REGION Network 10: EM - UnHolding State Complete
   RUNG wire#powerrail
      Contact( "EM02".PackML_Sts.Alarm.sts_UnHolding_SC )
      wire#w1
      Contact( "EM02".PackML_Sts.CM01.sts_UnHolding_SC )
      wire#w2
      Contact( "EM02".PackML_Sts.CM02.sts_UnHolding_SC )
      wire#w3
      Contact( "EM02".PackML_Sts.CM03.sts_UnHolding_SC )
      wire#w4
      Contact( "EM02".PackML_Sts.CM04.sts_UnHolding_SC )
      wire#w5
      Contact( "EM02".PackML_Sts.CM05.sts_UnHolding_SC )
      wire#w6
      Contact( "EM02".PackML_Sts.CM06.sts_UnHolding_SC )
      wire#w7
      Contact( "EM02".PackML_Sts.CM07.sts_UnHolding_SC )
      wire#w8
      Contact( "EM02".PackML_Sts.CM08.sts_UnHolding_SC )
      wire#w9
      Contact( "EM02".PackML_Sts.CM09.sts_UnHolding_SC )
      wire#w10
      Contact( "EM02".PackML_Sts.CM10.sts_UnHolding_SC )
      wire#w11
      Coil( "EM02".PackML_Sts.Unit.sts_UnHolding_SC )
   END_RUNG
   RUNG wire#powerrail
      I_Contact( "EM02".PackML_Sts.Alarm.moduleActive )
   END_RUNG wire#w1
   RUNG wire#w1
      I_Contact( "EM02".PackML_Sts.CM01.moduleActive )
   END_RUNG wire#w2
   RUNG wire#w2
      I_Contact( "EM02".PackML_Sts.CM02.moduleActive )
   END_RUNG wire#w3
   RUNG wire#w3
      I_Contact( "EM02".PackML_Sts.CM03.moduleActive )
   END_RUNG wire#w4
   RUNG wire#w4
      I_Contact( "EM02".PackML_Sts.CM04.moduleActive )
   END_RUNG wire#w5
   RUNG wire#w5
      I_Contact( "EM02".PackML_Sts.CM05.moduleActive )
   END_RUNG wire#w6
   RUNG wire#w6
      I_Contact( "EM02".PackML_Sts.CM06.moduleActive )
   END_RUNG wire#w7
   RUNG wire#w7
      I_Contact( "EM02".PackML_Sts.CM07.moduleActive )
   END_RUNG wire#w8
   RUNG wire#w8
      I_Contact( "EM02".PackML_Sts.CM08.moduleActive )
   END_RUNG wire#w9
   RUNG wire#w9
      I_Contact( "EM02".PackML_Sts.CM09.moduleActive )
   END_RUNG wire#w10
   RUNG wire#w10
      I_Contact( "EM02".PackML_Sts.CM10.moduleActive )
   END_RUNG wire#w11
   // the same network as SCL:
   "EM02".PackML_Sts.Unit.sts_UnHolding_SC := ("EM02".PackML_Sts.Alarm.sts_UnHolding_SC OR NOT "EM02".PackML_Sts.Alarm.moduleActive) AND ("EM02".PackML_Sts.CM01.sts_UnHolding_SC OR NOT "EM02".PackML_Sts.CM01.moduleActive) AND ("EM02".PackML_Sts.CM02.sts_UnHolding_SC OR NOT "EM02".PackML_Sts.CM02.moduleActive) AND ("EM02".PackML_Sts.CM03.sts_UnHolding_SC OR NOT "EM02".PackML_Sts.CM03.moduleActive) AND ("EM02".PackML_Sts.CM04.sts_UnHolding_SC OR NOT "EM02".PackML_Sts.CM04.moduleActive) AND ("EM02".PackML_Sts.CM05.sts_UnHolding_SC OR NOT "EM02".PackML_Sts.CM05.moduleActive) AND ("EM02".PackML_Sts.CM06.sts_UnHolding_SC OR NOT "EM02".PackML_Sts.CM06.moduleActive) AND ("EM02".PackML_Sts.CM07.sts_UnHolding_SC OR NOT "EM02".PackML_Sts.CM07.moduleActive) AND ("EM02".PackML_Sts.CM08.sts_UnHolding_SC OR NOT "EM02".PackML_Sts.CM08.moduleActive) AND ("EM02".PackML_Sts.CM09.sts_UnHolding_SC OR NOT "EM02".PackML_Sts.CM09.moduleActive) AND ("EM02".PackML_Sts.CM10.sts_UnHolding_SC OR NOT "EM02".PackML_Sts.CM10.moduleActive);
END_REGION

REGION Network 11: EM - Suspend Command
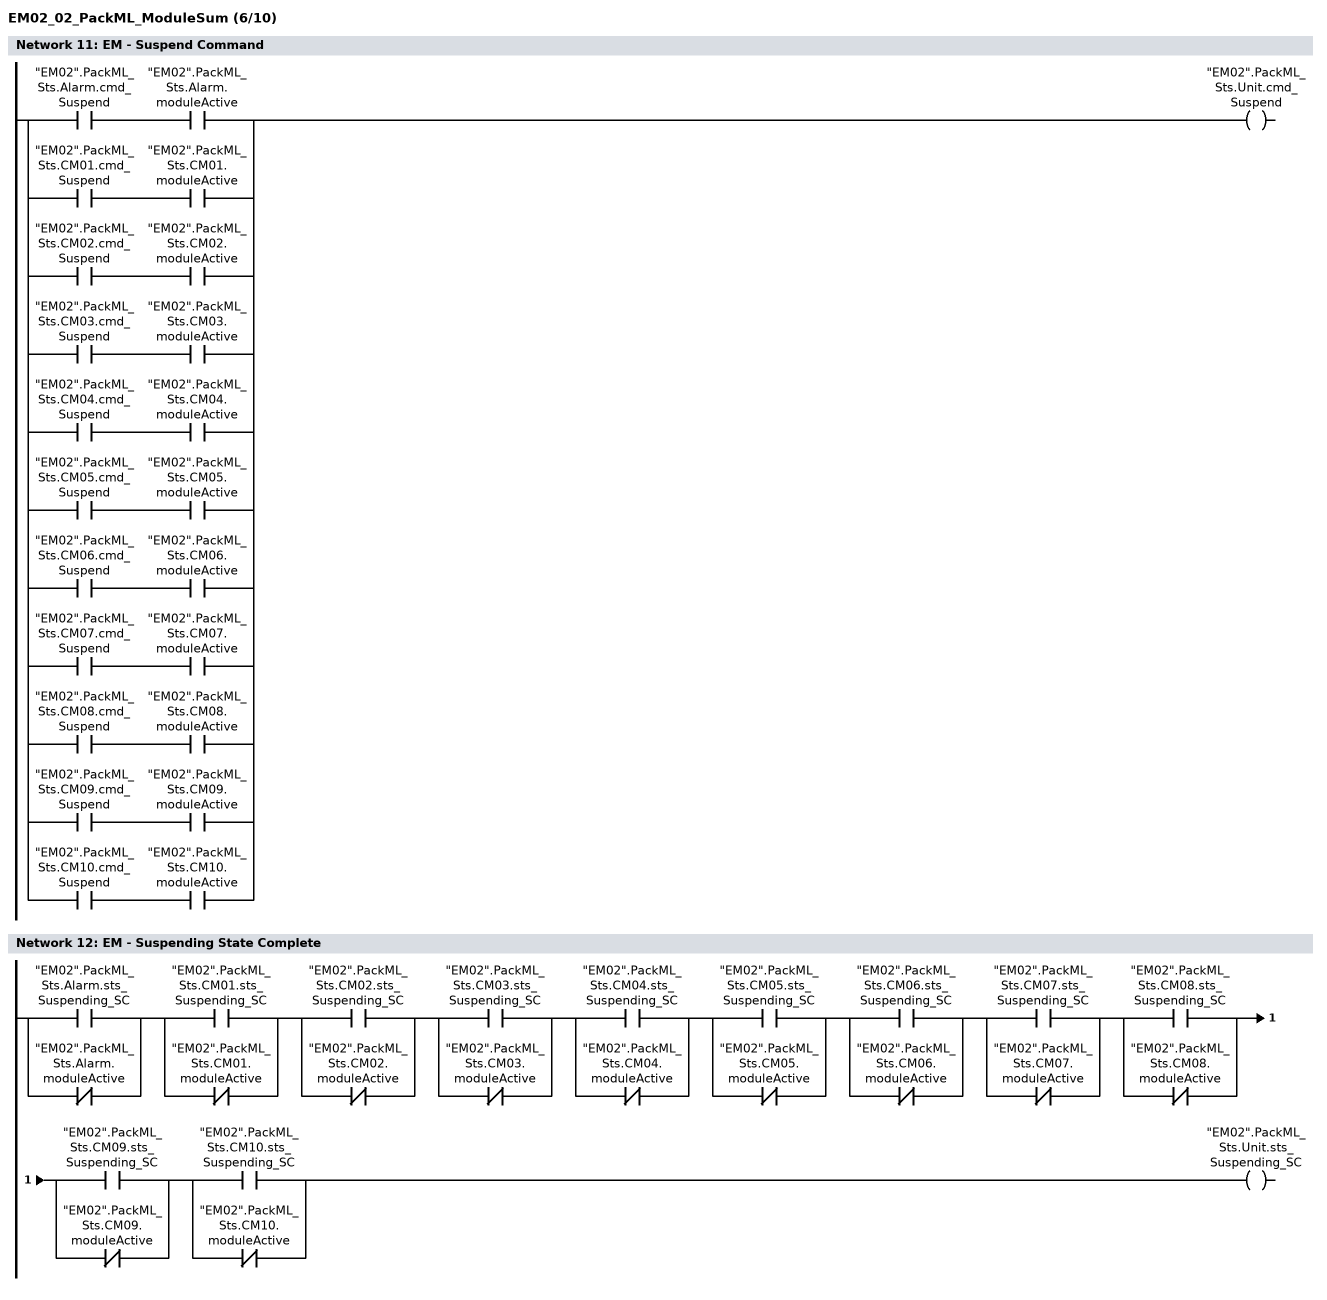
   RUNG wire#powerrail
      Contact( "EM02".PackML_Sts.Alarm.cmd_Suspend )
      Contact( "EM02".PackML_Sts.Alarm.moduleActive )
      wire#w1
      Coil( "EM02".PackML_Sts.Unit.cmd_Suspend )
   END_RUNG
   RUNG wire#powerrail
      Contact( "EM02".PackML_Sts.CM01.cmd_Suspend )
      Contact( "EM02".PackML_Sts.CM01.moduleActive )
   END_RUNG wire#w1
   RUNG wire#powerrail
      Contact( "EM02".PackML_Sts.CM02.cmd_Suspend )
      Contact( "EM02".PackML_Sts.CM02.moduleActive )
   END_RUNG wire#w1
   RUNG wire#powerrail
      Contact( "EM02".PackML_Sts.CM03.cmd_Suspend )
      Contact( "EM02".PackML_Sts.CM03.moduleActive )
   END_RUNG wire#w1
   RUNG wire#powerrail
      Contact( "EM02".PackML_Sts.CM04.cmd_Suspend )
      Contact( "EM02".PackML_Sts.CM04.moduleActive )
   END_RUNG wire#w1
   RUNG wire#powerrail
      Contact( "EM02".PackML_Sts.CM05.cmd_Suspend )
      Contact( "EM02".PackML_Sts.CM05.moduleActive )
   END_RUNG wire#w1
   RUNG wire#powerrail
      Contact( "EM02".PackML_Sts.CM06.cmd_Suspend )
      Contact( "EM02".PackML_Sts.CM06.moduleActive )
   END_RUNG wire#w1
   RUNG wire#powerrail
      Contact( "EM02".PackML_Sts.CM07.cmd_Suspend )
      Contact( "EM02".PackML_Sts.CM07.moduleActive )
   END_RUNG wire#w1
   RUNG wire#powerrail
      Contact( "EM02".PackML_Sts.CM08.cmd_Suspend )
      Contact( "EM02".PackML_Sts.CM08.moduleActive )
   END_RUNG wire#w1
   RUNG wire#powerrail
      Contact( "EM02".PackML_Sts.CM09.cmd_Suspend )
      Contact( "EM02".PackML_Sts.CM09.moduleActive )
   END_RUNG wire#w1
   RUNG wire#powerrail
      Contact( "EM02".PackML_Sts.CM10.cmd_Suspend )
      Contact( "EM02".PackML_Sts.CM10.moduleActive )
   END_RUNG wire#w1
   // the same network as SCL:
   "EM02".PackML_Sts.Unit.cmd_Suspend := ("EM02".PackML_Sts.Alarm.cmd_Suspend AND "EM02".PackML_Sts.Alarm.moduleActive) OR ("EM02".PackML_Sts.CM01.cmd_Suspend AND "EM02".PackML_Sts.CM01.moduleActive) OR ("EM02".PackML_Sts.CM02.cmd_Suspend AND "EM02".PackML_Sts.CM02.moduleActive) OR ("EM02".PackML_Sts.CM03.cmd_Suspend AND "EM02".PackML_Sts.CM03.moduleActive) OR ("EM02".PackML_Sts.CM04.cmd_Suspend AND "EM02".PackML_Sts.CM04.moduleActive) OR ("EM02".PackML_Sts.CM05.cmd_Suspend AND "EM02".PackML_Sts.CM05.moduleActive) OR ("EM02".PackML_Sts.CM06.cmd_Suspend AND "EM02".PackML_Sts.CM06.moduleActive) OR ("EM02".PackML_Sts.CM07.cmd_Suspend AND "EM02".PackML_Sts.CM07.moduleActive) OR ("EM02".PackML_Sts.CM08.cmd_Suspend AND "EM02".PackML_Sts.CM08.moduleActive) OR ("EM02".PackML_Sts.CM09.cmd_Suspend AND "EM02".PackML_Sts.CM09.moduleActive) OR ("EM02".PackML_Sts.CM10.cmd_Suspend AND "EM02".PackML_Sts.CM10.moduleActive);
END_REGION

REGION Network 12: EM - Suspending State Complete
   RUNG wire#powerrail
      Contact( "EM02".PackML_Sts.Alarm.sts_Suspending_SC )
      wire#w1
      Contact( "EM02".PackML_Sts.CM01.sts_Suspending_SC )
      wire#w2
      Contact( "EM02".PackML_Sts.CM02.sts_Suspending_SC )
      wire#w3
      Contact( "EM02".PackML_Sts.CM03.sts_Suspending_SC )
      wire#w4
      Contact( "EM02".PackML_Sts.CM04.sts_Suspending_SC )
      wire#w5
      Contact( "EM02".PackML_Sts.CM05.sts_Suspending_SC )
      wire#w6
      Contact( "EM02".PackML_Sts.CM06.sts_Suspending_SC )
      wire#w7
      Contact( "EM02".PackML_Sts.CM07.sts_Suspending_SC )
      wire#w8
      Contact( "EM02".PackML_Sts.CM08.sts_Suspending_SC )
      wire#w9
      Contact( "EM02".PackML_Sts.CM09.sts_Suspending_SC )
      wire#w10
      Contact( "EM02".PackML_Sts.CM10.sts_Suspending_SC )
      wire#w11
      Coil( "EM02".PackML_Sts.Unit.sts_Suspending_SC )
   END_RUNG
   RUNG wire#powerrail
      I_Contact( "EM02".PackML_Sts.Alarm.moduleActive )
   END_RUNG wire#w1
   RUNG wire#w1
      I_Contact( "EM02".PackML_Sts.CM01.moduleActive )
   END_RUNG wire#w2
   RUNG wire#w2
      I_Contact( "EM02".PackML_Sts.CM02.moduleActive )
   END_RUNG wire#w3
   RUNG wire#w3
      I_Contact( "EM02".PackML_Sts.CM03.moduleActive )
   END_RUNG wire#w4
   RUNG wire#w4
      I_Contact( "EM02".PackML_Sts.CM04.moduleActive )
   END_RUNG wire#w5
   RUNG wire#w5
      I_Contact( "EM02".PackML_Sts.CM05.moduleActive )
   END_RUNG wire#w6
   RUNG wire#w6
      I_Contact( "EM02".PackML_Sts.CM06.moduleActive )
   END_RUNG wire#w7
   RUNG wire#w7
      I_Contact( "EM02".PackML_Sts.CM07.moduleActive )
   END_RUNG wire#w8
   RUNG wire#w8
      I_Contact( "EM02".PackML_Sts.CM08.moduleActive )
   END_RUNG wire#w9
   RUNG wire#w9
      I_Contact( "EM02".PackML_Sts.CM09.moduleActive )
   END_RUNG wire#w10
   RUNG wire#w10
      I_Contact( "EM02".PackML_Sts.CM10.moduleActive )
   END_RUNG wire#w11
   // the same network as SCL:
   "EM02".PackML_Sts.Unit.sts_Suspending_SC := ("EM02".PackML_Sts.Alarm.sts_Suspending_SC OR NOT "EM02".PackML_Sts.Alarm.moduleActive) AND ("EM02".PackML_Sts.CM01.sts_Suspending_SC OR NOT "EM02".PackML_Sts.CM01.moduleActive) AND ("EM02".PackML_Sts.CM02.sts_Suspending_SC OR NOT "EM02".PackML_Sts.CM02.moduleActive) AND ("EM02".PackML_Sts.CM03.sts_Suspending_SC OR NOT "EM02".PackML_Sts.CM03.moduleActive) AND ("EM02".PackML_Sts.CM04.sts_Suspending_SC OR NOT "EM02".PackML_Sts.CM04.moduleActive) AND ("EM02".PackML_Sts.CM05.sts_Suspending_SC OR NOT "EM02".PackML_Sts.CM05.moduleActive) AND ("EM02".PackML_Sts.CM06.sts_Suspending_SC OR NOT "EM02".PackML_Sts.CM06.moduleActive) AND ("EM02".PackML_Sts.CM07.sts_Suspending_SC OR NOT "EM02".PackML_Sts.CM07.moduleActive) AND ("EM02".PackML_Sts.CM08.sts_Suspending_SC OR NOT "EM02".PackML_Sts.CM08.moduleActive) AND ("EM02".PackML_Sts.CM09.sts_Suspending_SC OR NOT "EM02".PackML_Sts.CM09.moduleActive) AND ("EM02".PackML_Sts.CM10.sts_Suspending_SC OR NOT "EM02".PackML_Sts.CM10.moduleActive);
END_REGION

REGION Network 13: EM - UnSuspend Command
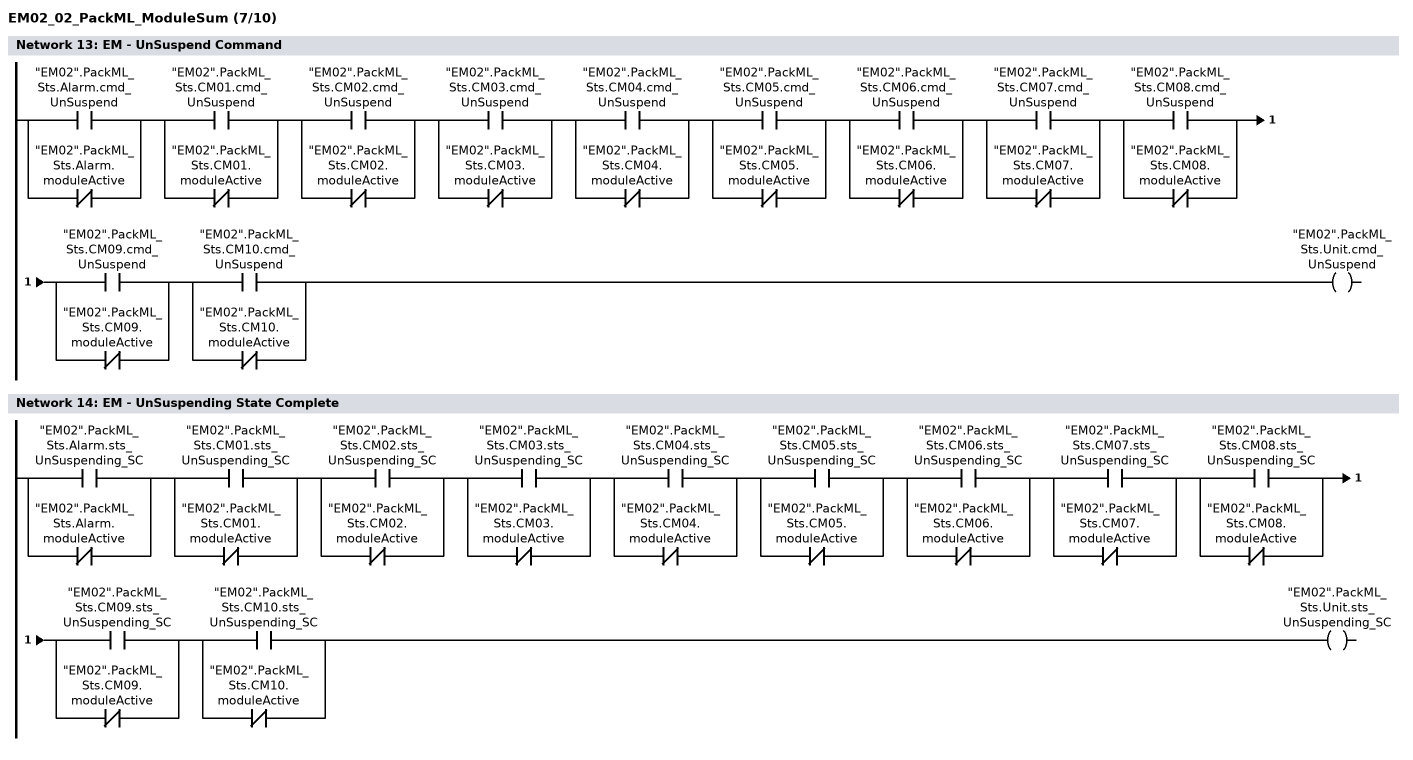
   RUNG wire#powerrail
      Contact( "EM02".PackML_Sts.Alarm.cmd_UnSuspend )
      wire#w1
      Contact( "EM02".PackML_Sts.CM01.cmd_UnSuspend )
      wire#w2
      Contact( "EM02".PackML_Sts.CM02.cmd_UnSuspend )
      wire#w3
      Contact( "EM02".PackML_Sts.CM03.cmd_UnSuspend )
      wire#w4
      Contact( "EM02".PackML_Sts.CM04.cmd_UnSuspend )
      wire#w5
      Contact( "EM02".PackML_Sts.CM05.cmd_UnSuspend )
      wire#w6
      Contact( "EM02".PackML_Sts.CM06.cmd_UnSuspend )
      wire#w7
      Contact( "EM02".PackML_Sts.CM07.cmd_UnSuspend )
      wire#w8
      Contact( "EM02".PackML_Sts.CM08.cmd_UnSuspend )
      wire#w9
      Contact( "EM02".PackML_Sts.CM09.cmd_UnSuspend )
      wire#w10
      Contact( "EM02".PackML_Sts.CM10.cmd_UnSuspend )
      wire#w11
      Coil( "EM02".PackML_Sts.Unit.cmd_UnSuspend )
   END_RUNG
   RUNG wire#powerrail
      I_Contact( "EM02".PackML_Sts.Alarm.moduleActive )
   END_RUNG wire#w1
   RUNG wire#w1
      I_Contact( "EM02".PackML_Sts.CM01.moduleActive )
   END_RUNG wire#w2
   RUNG wire#w2
      I_Contact( "EM02".PackML_Sts.CM02.moduleActive )
   END_RUNG wire#w3
   RUNG wire#w3
      I_Contact( "EM02".PackML_Sts.CM03.moduleActive )
   END_RUNG wire#w4
   RUNG wire#w4
      I_Contact( "EM02".PackML_Sts.CM04.moduleActive )
   END_RUNG wire#w5
   RUNG wire#w5
      I_Contact( "EM02".PackML_Sts.CM05.moduleActive )
   END_RUNG wire#w6
   RUNG wire#w6
      I_Contact( "EM02".PackML_Sts.CM06.moduleActive )
   END_RUNG wire#w7
   RUNG wire#w7
      I_Contact( "EM02".PackML_Sts.CM07.moduleActive )
   END_RUNG wire#w8
   RUNG wire#w8
      I_Contact( "EM02".PackML_Sts.CM08.moduleActive )
   END_RUNG wire#w9
   RUNG wire#w9
      I_Contact( "EM02".PackML_Sts.CM09.moduleActive )
   END_RUNG wire#w10
   RUNG wire#w10
      I_Contact( "EM02".PackML_Sts.CM10.moduleActive )
   END_RUNG wire#w11
   // the same network as SCL:
   "EM02".PackML_Sts.Unit.cmd_UnSuspend := ("EM02".PackML_Sts.Alarm.cmd_UnSuspend OR NOT "EM02".PackML_Sts.Alarm.moduleActive) AND ("EM02".PackML_Sts.CM01.cmd_UnSuspend OR NOT "EM02".PackML_Sts.CM01.moduleActive) AND ("EM02".PackML_Sts.CM02.cmd_UnSuspend OR NOT "EM02".PackML_Sts.CM02.moduleActive) AND ("EM02".PackML_Sts.CM03.cmd_UnSuspend OR NOT "EM02".PackML_Sts.CM03.moduleActive) AND ("EM02".PackML_Sts.CM04.cmd_UnSuspend OR NOT "EM02".PackML_Sts.CM04.moduleActive) AND ("EM02".PackML_Sts.CM05.cmd_UnSuspend OR NOT "EM02".PackML_Sts.CM05.moduleActive) AND ("EM02".PackML_Sts.CM06.cmd_UnSuspend OR NOT "EM02".PackML_Sts.CM06.moduleActive) AND ("EM02".PackML_Sts.CM07.cmd_UnSuspend OR NOT "EM02".PackML_Sts.CM07.moduleActive) AND ("EM02".PackML_Sts.CM08.cmd_UnSuspend OR NOT "EM02".PackML_Sts.CM08.moduleActive) AND ("EM02".PackML_Sts.CM09.cmd_UnSuspend OR NOT "EM02".PackML_Sts.CM09.moduleActive) AND ("EM02".PackML_Sts.CM10.cmd_UnSuspend OR NOT "EM02".PackML_Sts.CM10.moduleActive);
END_REGION

REGION Network 14: EM - UnSuspending State Complete
   RUNG wire#powerrail
      Contact( "EM02".PackML_Sts.Alarm.sts_UnSuspending_SC )
      wire#w1
      Contact( "EM02".PackML_Sts.CM01.sts_UnSuspending_SC )
      wire#w2
      Contact( "EM02".PackML_Sts.CM02.sts_UnSuspending_SC )
      wire#w3
      Contact( "EM02".PackML_Sts.CM03.sts_UnSuspending_SC )
      wire#w4
      Contact( "EM02".PackML_Sts.CM04.sts_UnSuspending_SC )
      wire#w5
      Contact( "EM02".PackML_Sts.CM05.sts_UnSuspending_SC )
      wire#w6
      Contact( "EM02".PackML_Sts.CM06.sts_UnSuspending_SC )
      wire#w7
      Contact( "EM02".PackML_Sts.CM07.sts_UnSuspending_SC )
      wire#w8
      Contact( "EM02".PackML_Sts.CM08.sts_UnSuspending_SC )
      wire#w9
      Contact( "EM02".PackML_Sts.CM09.sts_UnSuspending_SC )
      wire#w10
      Contact( "EM02".PackML_Sts.CM10.sts_UnSuspending_SC )
      wire#w11
      Coil( "EM02".PackML_Sts.Unit.sts_UnSuspending_SC )
   END_RUNG
   RUNG wire#powerrail
      I_Contact( "EM02".PackML_Sts.Alarm.moduleActive )
   END_RUNG wire#w1
   RUNG wire#w1
      I_Contact( "EM02".PackML_Sts.CM01.moduleActive )
   END_RUNG wire#w2
   RUNG wire#w2
      I_Contact( "EM02".PackML_Sts.CM02.moduleActive )
   END_RUNG wire#w3
   RUNG wire#w3
      I_Contact( "EM02".PackML_Sts.CM03.moduleActive )
   END_RUNG wire#w4
   RUNG wire#w4
      I_Contact( "EM02".PackML_Sts.CM04.moduleActive )
   END_RUNG wire#w5
   RUNG wire#w5
      I_Contact( "EM02".PackML_Sts.CM05.moduleActive )
   END_RUNG wire#w6
   RUNG wire#w6
      I_Contact( "EM02".PackML_Sts.CM06.moduleActive )
   END_RUNG wire#w7
   RUNG wire#w7
      I_Contact( "EM02".PackML_Sts.CM07.moduleActive )
   END_RUNG wire#w8
   RUNG wire#w8
      I_Contact( "EM02".PackML_Sts.CM08.moduleActive )
   END_RUNG wire#w9
   RUNG wire#w9
      I_Contact( "EM02".PackML_Sts.CM09.moduleActive )
   END_RUNG wire#w10
   RUNG wire#w10
      I_Contact( "EM02".PackML_Sts.CM10.moduleActive )
   END_RUNG wire#w11
   // the same network as SCL:
   "EM02".PackML_Sts.Unit.sts_UnSuspending_SC := ("EM02".PackML_Sts.Alarm.sts_UnSuspending_SC OR NOT "EM02".PackML_Sts.Alarm.moduleActive) AND ("EM02".PackML_Sts.CM01.sts_UnSuspending_SC OR NOT "EM02".PackML_Sts.CM01.moduleActive) AND ("EM02".PackML_Sts.CM02.sts_UnSuspending_SC OR NOT "EM02".PackML_Sts.CM02.moduleActive) AND ("EM02".PackML_Sts.CM03.sts_UnSuspending_SC OR NOT "EM02".PackML_Sts.CM03.moduleActive) AND ("EM02".PackML_Sts.CM04.sts_UnSuspending_SC OR NOT "EM02".PackML_Sts.CM04.moduleActive) AND ("EM02".PackML_Sts.CM05.sts_UnSuspending_SC OR NOT "EM02".PackML_Sts.CM05.moduleActive) AND ("EM02".PackML_Sts.CM06.sts_UnSuspending_SC OR NOT "EM02".PackML_Sts.CM06.moduleActive) AND ("EM02".PackML_Sts.CM07.sts_UnSuspending_SC OR NOT "EM02".PackML_Sts.CM07.moduleActive) AND ("EM02".PackML_Sts.CM08.sts_UnSuspending_SC OR NOT "EM02".PackML_Sts.CM08.moduleActive) AND ("EM02".PackML_Sts.CM09.sts_UnSuspending_SC OR NOT "EM02".PackML_Sts.CM09.moduleActive) AND ("EM02".PackML_Sts.CM10.sts_UnSuspending_SC OR NOT "EM02".PackML_Sts.CM10.moduleActive);
END_REGION

REGION Network 15: EM - Abort Command
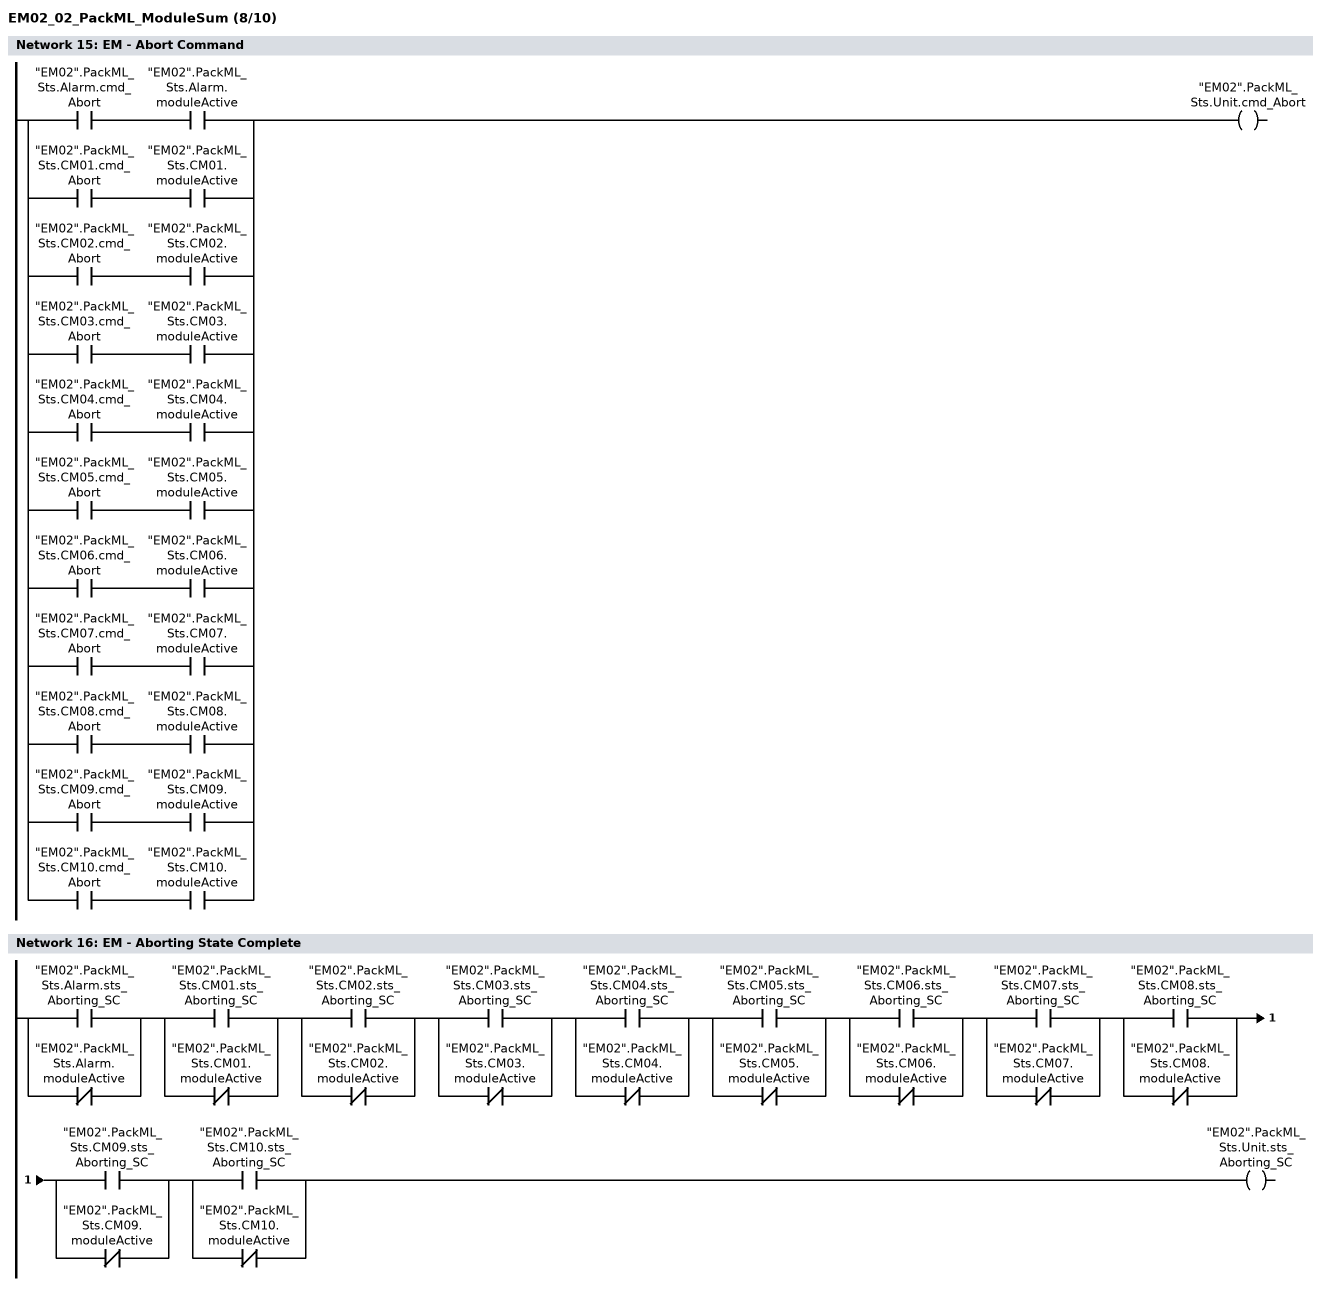
   RUNG wire#powerrail
      Contact( "EM02".PackML_Sts.Alarm.cmd_Abort )
      Contact( "EM02".PackML_Sts.Alarm.moduleActive )
      wire#w1
      Coil( "EM02".PackML_Sts.Unit.cmd_Abort )
   END_RUNG
   RUNG wire#powerrail
      Contact( "EM02".PackML_Sts.CM01.cmd_Abort )
      Contact( "EM02".PackML_Sts.CM01.moduleActive )
   END_RUNG wire#w1
   RUNG wire#powerrail
      Contact( "EM02".PackML_Sts.CM02.cmd_Abort )
      Contact( "EM02".PackML_Sts.CM02.moduleActive )
   END_RUNG wire#w1
   RUNG wire#powerrail
      Contact( "EM02".PackML_Sts.CM03.cmd_Abort )
      Contact( "EM02".PackML_Sts.CM03.moduleActive )
   END_RUNG wire#w1
   RUNG wire#powerrail
      Contact( "EM02".PackML_Sts.CM04.cmd_Abort )
      Contact( "EM02".PackML_Sts.CM04.moduleActive )
   END_RUNG wire#w1
   RUNG wire#powerrail
      Contact( "EM02".PackML_Sts.CM05.cmd_Abort )
      Contact( "EM02".PackML_Sts.CM05.moduleActive )
   END_RUNG wire#w1
   RUNG wire#powerrail
      Contact( "EM02".PackML_Sts.CM06.cmd_Abort )
      Contact( "EM02".PackML_Sts.CM06.moduleActive )
   END_RUNG wire#w1
   RUNG wire#powerrail
      Contact( "EM02".PackML_Sts.CM07.cmd_Abort )
      Contact( "EM02".PackML_Sts.CM07.moduleActive )
   END_RUNG wire#w1
   RUNG wire#powerrail
      Contact( "EM02".PackML_Sts.CM08.cmd_Abort )
      Contact( "EM02".PackML_Sts.CM08.moduleActive )
   END_RUNG wire#w1
   RUNG wire#powerrail
      Contact( "EM02".PackML_Sts.CM09.cmd_Abort )
      Contact( "EM02".PackML_Sts.CM09.moduleActive )
   END_RUNG wire#w1
   RUNG wire#powerrail
      Contact( "EM02".PackML_Sts.CM10.cmd_Abort )
      Contact( "EM02".PackML_Sts.CM10.moduleActive )
   END_RUNG wire#w1
   // the same network as SCL:
   "EM02".PackML_Sts.Unit.cmd_Abort := ("EM02".PackML_Sts.Alarm.cmd_Abort AND "EM02".PackML_Sts.Alarm.moduleActive) OR ("EM02".PackML_Sts.CM01.cmd_Abort AND "EM02".PackML_Sts.CM01.moduleActive) OR ("EM02".PackML_Sts.CM02.cmd_Abort AND "EM02".PackML_Sts.CM02.moduleActive) OR ("EM02".PackML_Sts.CM03.cmd_Abort AND "EM02".PackML_Sts.CM03.moduleActive) OR ("EM02".PackML_Sts.CM04.cmd_Abort AND "EM02".PackML_Sts.CM04.moduleActive) OR ("EM02".PackML_Sts.CM05.cmd_Abort AND "EM02".PackML_Sts.CM05.moduleActive) OR ("EM02".PackML_Sts.CM06.cmd_Abort AND "EM02".PackML_Sts.CM06.moduleActive) OR ("EM02".PackML_Sts.CM07.cmd_Abort AND "EM02".PackML_Sts.CM07.moduleActive) OR ("EM02".PackML_Sts.CM08.cmd_Abort AND "EM02".PackML_Sts.CM08.moduleActive) OR ("EM02".PackML_Sts.CM09.cmd_Abort AND "EM02".PackML_Sts.CM09.moduleActive) OR ("EM02".PackML_Sts.CM10.cmd_Abort AND "EM02".PackML_Sts.CM10.moduleActive);
END_REGION

REGION Network 16: EM - Aborting State Complete
   RUNG wire#powerrail
      Contact( "EM02".PackML_Sts.Alarm.sts_Aborting_SC )
      wire#w1
      Contact( "EM02".PackML_Sts.CM01.sts_Aborting_SC )
      wire#w2
      Contact( "EM02".PackML_Sts.CM02.sts_Aborting_SC )
      wire#w3
      Contact( "EM02".PackML_Sts.CM03.sts_Aborting_SC )
      wire#w4
      Contact( "EM02".PackML_Sts.CM04.sts_Aborting_SC )
      wire#w5
      Contact( "EM02".PackML_Sts.CM05.sts_Aborting_SC )
      wire#w6
      Contact( "EM02".PackML_Sts.CM06.sts_Aborting_SC )
      wire#w7
      Contact( "EM02".PackML_Sts.CM07.sts_Aborting_SC )
      wire#w8
      Contact( "EM02".PackML_Sts.CM08.sts_Aborting_SC )
      wire#w9
      Contact( "EM02".PackML_Sts.CM09.sts_Aborting_SC )
      wire#w10
      Contact( "EM02".PackML_Sts.CM10.sts_Aborting_SC )
      wire#w11
      Coil( "EM02".PackML_Sts.Unit.sts_Aborting_SC )
   END_RUNG
   RUNG wire#powerrail
      I_Contact( "EM02".PackML_Sts.Alarm.moduleActive )
   END_RUNG wire#w1
   RUNG wire#w1
      I_Contact( "EM02".PackML_Sts.CM01.moduleActive )
   END_RUNG wire#w2
   RUNG wire#w2
      I_Contact( "EM02".PackML_Sts.CM02.moduleActive )
   END_RUNG wire#w3
   RUNG wire#w3
      I_Contact( "EM02".PackML_Sts.CM03.moduleActive )
   END_RUNG wire#w4
   RUNG wire#w4
      I_Contact( "EM02".PackML_Sts.CM04.moduleActive )
   END_RUNG wire#w5
   RUNG wire#w5
      I_Contact( "EM02".PackML_Sts.CM05.moduleActive )
   END_RUNG wire#w6
   RUNG wire#w6
      I_Contact( "EM02".PackML_Sts.CM06.moduleActive )
   END_RUNG wire#w7
   RUNG wire#w7
      I_Contact( "EM02".PackML_Sts.CM07.moduleActive )
   END_RUNG wire#w8
   RUNG wire#w8
      I_Contact( "EM02".PackML_Sts.CM08.moduleActive )
   END_RUNG wire#w9
   RUNG wire#w9
      I_Contact( "EM02".PackML_Sts.CM09.moduleActive )
   END_RUNG wire#w10
   RUNG wire#w10
      I_Contact( "EM02".PackML_Sts.CM10.moduleActive )
   END_RUNG wire#w11
   // the same network as SCL:
   "EM02".PackML_Sts.Unit.sts_Aborting_SC := ("EM02".PackML_Sts.Alarm.sts_Aborting_SC OR NOT "EM02".PackML_Sts.Alarm.moduleActive) AND ("EM02".PackML_Sts.CM01.sts_Aborting_SC OR NOT "EM02".PackML_Sts.CM01.moduleActive) AND ("EM02".PackML_Sts.CM02.sts_Aborting_SC OR NOT "EM02".PackML_Sts.CM02.moduleActive) AND ("EM02".PackML_Sts.CM03.sts_Aborting_SC OR NOT "EM02".PackML_Sts.CM03.moduleActive) AND ("EM02".PackML_Sts.CM04.sts_Aborting_SC OR NOT "EM02".PackML_Sts.CM04.moduleActive) AND ("EM02".PackML_Sts.CM05.sts_Aborting_SC OR NOT "EM02".PackML_Sts.CM05.moduleActive) AND ("EM02".PackML_Sts.CM06.sts_Aborting_SC OR NOT "EM02".PackML_Sts.CM06.moduleActive) AND ("EM02".PackML_Sts.CM07.sts_Aborting_SC OR NOT "EM02".PackML_Sts.CM07.moduleActive) AND ("EM02".PackML_Sts.CM08.sts_Aborting_SC OR NOT "EM02".PackML_Sts.CM08.moduleActive) AND ("EM02".PackML_Sts.CM09.sts_Aborting_SC OR NOT "EM02".PackML_Sts.CM09.moduleActive) AND ("EM02".PackML_Sts.CM10.sts_Aborting_SC OR NOT "EM02".PackML_Sts.CM10.moduleActive);
END_REGION

REGION Network 17: EM - Clear Command
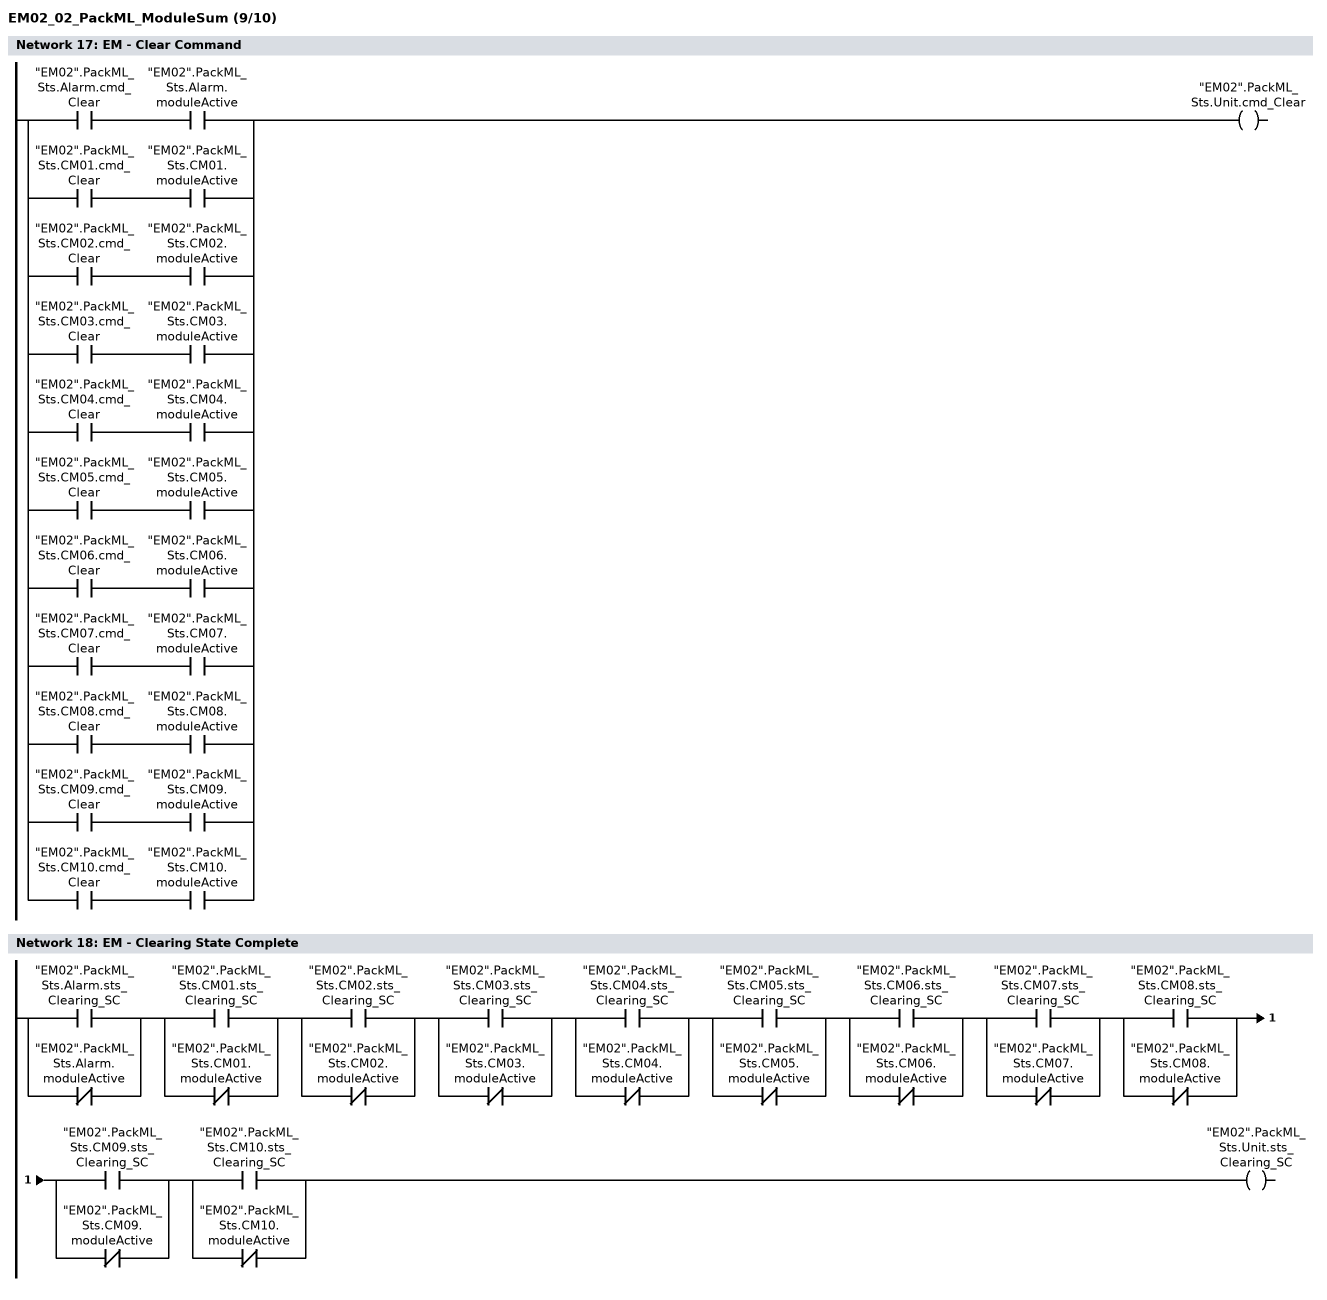
   RUNG wire#powerrail
      Contact( "EM02".PackML_Sts.Alarm.cmd_Clear )
      Contact( "EM02".PackML_Sts.Alarm.moduleActive )
      wire#w1
      Coil( "EM02".PackML_Sts.Unit.cmd_Clear )
   END_RUNG
   RUNG wire#powerrail
      Contact( "EM02".PackML_Sts.CM01.cmd_Clear )
      Contact( "EM02".PackML_Sts.CM01.moduleActive )
   END_RUNG wire#w1
   RUNG wire#powerrail
      Contact( "EM02".PackML_Sts.CM02.cmd_Clear )
      Contact( "EM02".PackML_Sts.CM02.moduleActive )
   END_RUNG wire#w1
   RUNG wire#powerrail
      Contact( "EM02".PackML_Sts.CM03.cmd_Clear )
      Contact( "EM02".PackML_Sts.CM03.moduleActive )
   END_RUNG wire#w1
   RUNG wire#powerrail
      Contact( "EM02".PackML_Sts.CM04.cmd_Clear )
      Contact( "EM02".PackML_Sts.CM04.moduleActive )
   END_RUNG wire#w1
   RUNG wire#powerrail
      Contact( "EM02".PackML_Sts.CM05.cmd_Clear )
      Contact( "EM02".PackML_Sts.CM05.moduleActive )
   END_RUNG wire#w1
   RUNG wire#powerrail
      Contact( "EM02".PackML_Sts.CM06.cmd_Clear )
      Contact( "EM02".PackML_Sts.CM06.moduleActive )
   END_RUNG wire#w1
   RUNG wire#powerrail
      Contact( "EM02".PackML_Sts.CM07.cmd_Clear )
      Contact( "EM02".PackML_Sts.CM07.moduleActive )
   END_RUNG wire#w1
   RUNG wire#powerrail
      Contact( "EM02".PackML_Sts.CM08.cmd_Clear )
      Contact( "EM02".PackML_Sts.CM08.moduleActive )
   END_RUNG wire#w1
   RUNG wire#powerrail
      Contact( "EM02".PackML_Sts.CM09.cmd_Clear )
      Contact( "EM02".PackML_Sts.CM09.moduleActive )
   END_RUNG wire#w1
   RUNG wire#powerrail
      Contact( "EM02".PackML_Sts.CM10.cmd_Clear )
      Contact( "EM02".PackML_Sts.CM10.moduleActive )
   END_RUNG wire#w1
   // the same network as SCL:
   "EM02".PackML_Sts.Unit.cmd_Clear := ("EM02".PackML_Sts.Alarm.cmd_Clear AND "EM02".PackML_Sts.Alarm.moduleActive) OR ("EM02".PackML_Sts.CM01.cmd_Clear AND "EM02".PackML_Sts.CM01.moduleActive) OR ("EM02".PackML_Sts.CM02.cmd_Clear AND "EM02".PackML_Sts.CM02.moduleActive) OR ("EM02".PackML_Sts.CM03.cmd_Clear AND "EM02".PackML_Sts.CM03.moduleActive) OR ("EM02".PackML_Sts.CM04.cmd_Clear AND "EM02".PackML_Sts.CM04.moduleActive) OR ("EM02".PackML_Sts.CM05.cmd_Clear AND "EM02".PackML_Sts.CM05.moduleActive) OR ("EM02".PackML_Sts.CM06.cmd_Clear AND "EM02".PackML_Sts.CM06.moduleActive) OR ("EM02".PackML_Sts.CM07.cmd_Clear AND "EM02".PackML_Sts.CM07.moduleActive) OR ("EM02".PackML_Sts.CM08.cmd_Clear AND "EM02".PackML_Sts.CM08.moduleActive) OR ("EM02".PackML_Sts.CM09.cmd_Clear AND "EM02".PackML_Sts.CM09.moduleActive) OR ("EM02".PackML_Sts.CM10.cmd_Clear AND "EM02".PackML_Sts.CM10.moduleActive);
END_REGION

REGION Network 18: EM - Clearing State Complete
   RUNG wire#powerrail
      Contact( "EM02".PackML_Sts.Alarm.sts_Clearing_SC )
      wire#w1
      Contact( "EM02".PackML_Sts.CM01.sts_Clearing_SC )
      wire#w2
      Contact( "EM02".PackML_Sts.CM02.sts_Clearing_SC )
      wire#w3
      Contact( "EM02".PackML_Sts.CM03.sts_Clearing_SC )
      wire#w4
      Contact( "EM02".PackML_Sts.CM04.sts_Clearing_SC )
      wire#w5
      Contact( "EM02".PackML_Sts.CM05.sts_Clearing_SC )
      wire#w6
      Contact( "EM02".PackML_Sts.CM06.sts_Clearing_SC )
      wire#w7
      Contact( "EM02".PackML_Sts.CM07.sts_Clearing_SC )
      wire#w8
      Contact( "EM02".PackML_Sts.CM08.sts_Clearing_SC )
      wire#w9
      Contact( "EM02".PackML_Sts.CM09.sts_Clearing_SC )
      wire#w10
      Contact( "EM02".PackML_Sts.CM10.sts_Clearing_SC )
      wire#w11
      Coil( "EM02".PackML_Sts.Unit.sts_Clearing_SC )
   END_RUNG
   RUNG wire#powerrail
      I_Contact( "EM02".PackML_Sts.Alarm.moduleActive )
   END_RUNG wire#w1
   RUNG wire#w1
      I_Contact( "EM02".PackML_Sts.CM01.moduleActive )
   END_RUNG wire#w2
   RUNG wire#w2
      I_Contact( "EM02".PackML_Sts.CM02.moduleActive )
   END_RUNG wire#w3
   RUNG wire#w3
      I_Contact( "EM02".PackML_Sts.CM03.moduleActive )
   END_RUNG wire#w4
   RUNG wire#w4
      I_Contact( "EM02".PackML_Sts.CM04.moduleActive )
   END_RUNG wire#w5
   RUNG wire#w5
      I_Contact( "EM02".PackML_Sts.CM05.moduleActive )
   END_RUNG wire#w6
   RUNG wire#w6
      I_Contact( "EM02".PackML_Sts.CM06.moduleActive )
   END_RUNG wire#w7
   RUNG wire#w7
      I_Contact( "EM02".PackML_Sts.CM07.moduleActive )
   END_RUNG wire#w8
   RUNG wire#w8
      I_Contact( "EM02".PackML_Sts.CM08.moduleActive )
   END_RUNG wire#w9
   RUNG wire#w9
      I_Contact( "EM02".PackML_Sts.CM09.moduleActive )
   END_RUNG wire#w10
   RUNG wire#w10
      I_Contact( "EM02".PackML_Sts.CM10.moduleActive )
   END_RUNG wire#w11
   // the same network as SCL:
   "EM02".PackML_Sts.Unit.sts_Clearing_SC := ("EM02".PackML_Sts.Alarm.sts_Clearing_SC OR NOT "EM02".PackML_Sts.Alarm.moduleActive) AND ("EM02".PackML_Sts.CM01.sts_Clearing_SC OR NOT "EM02".PackML_Sts.CM01.moduleActive) AND ("EM02".PackML_Sts.CM02.sts_Clearing_SC OR NOT "EM02".PackML_Sts.CM02.moduleActive) AND ("EM02".PackML_Sts.CM03.sts_Clearing_SC OR NOT "EM02".PackML_Sts.CM03.moduleActive) AND ("EM02".PackML_Sts.CM04.sts_Clearing_SC OR NOT "EM02".PackML_Sts.CM04.moduleActive) AND ("EM02".PackML_Sts.CM05.sts_Clearing_SC OR NOT "EM02".PackML_Sts.CM05.moduleActive) AND ("EM02".PackML_Sts.CM06.sts_Clearing_SC OR NOT "EM02".PackML_Sts.CM06.moduleActive) AND ("EM02".PackML_Sts.CM07.sts_Clearing_SC OR NOT "EM02".PackML_Sts.CM07.moduleActive) AND ("EM02".PackML_Sts.CM08.sts_Clearing_SC OR NOT "EM02".PackML_Sts.CM08.moduleActive) AND ("EM02".PackML_Sts.CM09.sts_Clearing_SC OR NOT "EM02".PackML_Sts.CM09.moduleActive) AND ("EM02".PackML_Sts.CM10.sts_Clearing_SC OR NOT "EM02".PackML_Sts.CM10.moduleActive);
END_REGION

REGION Network 19: EM - Execute State Complete
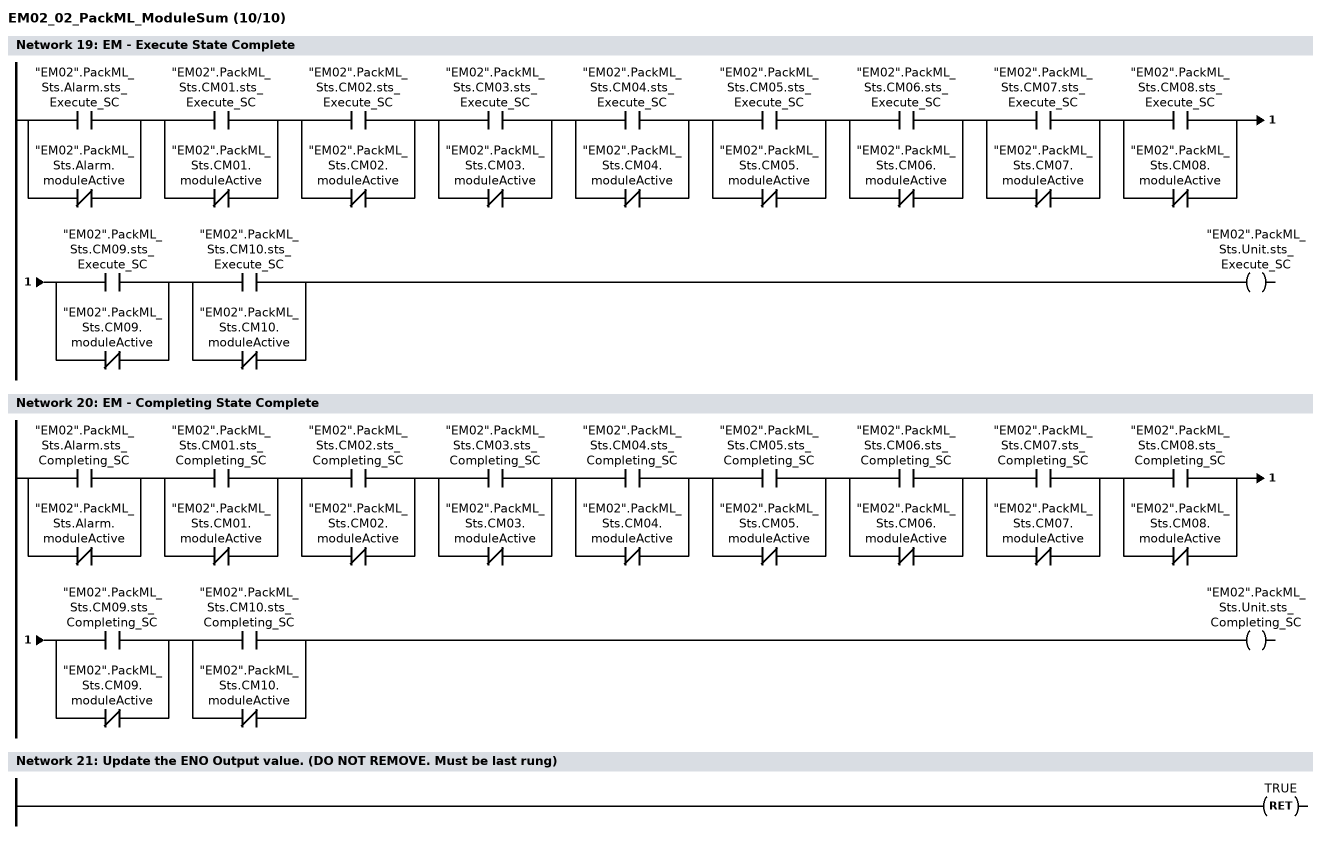
   RUNG wire#powerrail
      Contact( "EM02".PackML_Sts.Alarm.sts_Execute_SC )
      wire#w1
      Contact( "EM02".PackML_Sts.CM01.sts_Execute_SC )
      wire#w2
      Contact( "EM02".PackML_Sts.CM02.sts_Execute_SC )
      wire#w3
      Contact( "EM02".PackML_Sts.CM03.sts_Execute_SC )
      wire#w4
      Contact( "EM02".PackML_Sts.CM04.sts_Execute_SC )
      wire#w5
      Contact( "EM02".PackML_Sts.CM05.sts_Execute_SC )
      wire#w6
      Contact( "EM02".PackML_Sts.CM06.sts_Execute_SC )
      wire#w7
      Contact( "EM02".PackML_Sts.CM07.sts_Execute_SC )
      wire#w8
      Contact( "EM02".PackML_Sts.CM08.sts_Execute_SC )
      wire#w9
      Contact( "EM02".PackML_Sts.CM09.sts_Execute_SC )
      wire#w10
      Contact( "EM02".PackML_Sts.CM10.sts_Execute_SC )
      wire#w11
      Coil( "EM02".PackML_Sts.Unit.sts_Execute_SC )
   END_RUNG
   RUNG wire#powerrail
      I_Contact( "EM02".PackML_Sts.Alarm.moduleActive )
   END_RUNG wire#w1
   RUNG wire#w1
      I_Contact( "EM02".PackML_Sts.CM01.moduleActive )
   END_RUNG wire#w2
   RUNG wire#w2
      I_Contact( "EM02".PackML_Sts.CM02.moduleActive )
   END_RUNG wire#w3
   RUNG wire#w3
      I_Contact( "EM02".PackML_Sts.CM03.moduleActive )
   END_RUNG wire#w4
   RUNG wire#w4
      I_Contact( "EM02".PackML_Sts.CM04.moduleActive )
   END_RUNG wire#w5
   RUNG wire#w5
      I_Contact( "EM02".PackML_Sts.CM05.moduleActive )
   END_RUNG wire#w6
   RUNG wire#w6
      I_Contact( "EM02".PackML_Sts.CM06.moduleActive )
   END_RUNG wire#w7
   RUNG wire#w7
      I_Contact( "EM02".PackML_Sts.CM07.moduleActive )
   END_RUNG wire#w8
   RUNG wire#w8
      I_Contact( "EM02".PackML_Sts.CM08.moduleActive )
   END_RUNG wire#w9
   RUNG wire#w9
      I_Contact( "EM02".PackML_Sts.CM09.moduleActive )
   END_RUNG wire#w10
   RUNG wire#w10
      I_Contact( "EM02".PackML_Sts.CM10.moduleActive )
   END_RUNG wire#w11
   // the same network as SCL:
   "EM02".PackML_Sts.Unit.sts_Execute_SC := ("EM02".PackML_Sts.Alarm.sts_Execute_SC OR NOT "EM02".PackML_Sts.Alarm.moduleActive) AND ("EM02".PackML_Sts.CM01.sts_Execute_SC OR NOT "EM02".PackML_Sts.CM01.moduleActive) AND ("EM02".PackML_Sts.CM02.sts_Execute_SC OR NOT "EM02".PackML_Sts.CM02.moduleActive) AND ("EM02".PackML_Sts.CM03.sts_Execute_SC OR NOT "EM02".PackML_Sts.CM03.moduleActive) AND ("EM02".PackML_Sts.CM04.sts_Execute_SC OR NOT "EM02".PackML_Sts.CM04.moduleActive) AND ("EM02".PackML_Sts.CM05.sts_Execute_SC OR NOT "EM02".PackML_Sts.CM05.moduleActive) AND ("EM02".PackML_Sts.CM06.sts_Execute_SC OR NOT "EM02".PackML_Sts.CM06.moduleActive) AND ("EM02".PackML_Sts.CM07.sts_Execute_SC OR NOT "EM02".PackML_Sts.CM07.moduleActive) AND ("EM02".PackML_Sts.CM08.sts_Execute_SC OR NOT "EM02".PackML_Sts.CM08.moduleActive) AND ("EM02".PackML_Sts.CM09.sts_Execute_SC OR NOT "EM02".PackML_Sts.CM09.moduleActive) AND ("EM02".PackML_Sts.CM10.sts_Execute_SC OR NOT "EM02".PackML_Sts.CM10.moduleActive);
END_REGION

REGION Network 20: EM - Completing State Complete
   RUNG wire#powerrail
      Contact( "EM02".PackML_Sts.Alarm.sts_Completing_SC )
      wire#w1
      Contact( "EM02".PackML_Sts.CM01.sts_Completing_SC )
      wire#w2
      Contact( "EM02".PackML_Sts.CM02.sts_Completing_SC )
      wire#w3
      Contact( "EM02".PackML_Sts.CM03.sts_Completing_SC )
      wire#w4
      Contact( "EM02".PackML_Sts.CM04.sts_Completing_SC )
      wire#w5
      Contact( "EM02".PackML_Sts.CM05.sts_Completing_SC )
      wire#w6
      Contact( "EM02".PackML_Sts.CM06.sts_Completing_SC )
      wire#w7
      Contact( "EM02".PackML_Sts.CM07.sts_Completing_SC )
      wire#w8
      Contact( "EM02".PackML_Sts.CM08.sts_Completing_SC )
      wire#w9
      Contact( "EM02".PackML_Sts.CM09.sts_Completing_SC )
      wire#w10
      Contact( "EM02".PackML_Sts.CM10.sts_Completing_SC )
      wire#w11
      Coil( "EM02".PackML_Sts.Unit.sts_Completing_SC )
   END_RUNG
   RUNG wire#powerrail
      I_Contact( "EM02".PackML_Sts.Alarm.moduleActive )
   END_RUNG wire#w1
   RUNG wire#w1
      I_Contact( "EM02".PackML_Sts.CM01.moduleActive )
   END_RUNG wire#w2
   RUNG wire#w2
      I_Contact( "EM02".PackML_Sts.CM02.moduleActive )
   END_RUNG wire#w3
   RUNG wire#w3
      I_Contact( "EM02".PackML_Sts.CM03.moduleActive )
   END_RUNG wire#w4
   RUNG wire#w4
      I_Contact( "EM02".PackML_Sts.CM04.moduleActive )
   END_RUNG wire#w5
   RUNG wire#w5
      I_Contact( "EM02".PackML_Sts.CM05.moduleActive )
   END_RUNG wire#w6
   RUNG wire#w6
      I_Contact( "EM02".PackML_Sts.CM06.moduleActive )
   END_RUNG wire#w7
   RUNG wire#w7
      I_Contact( "EM02".PackML_Sts.CM07.moduleActive )
   END_RUNG wire#w8
   RUNG wire#w8
      I_Contact( "EM02".PackML_Sts.CM08.moduleActive )
   END_RUNG wire#w9
   RUNG wire#w9
      I_Contact( "EM02".PackML_Sts.CM09.moduleActive )
   END_RUNG wire#w10
   RUNG wire#w10
      I_Contact( "EM02".PackML_Sts.CM10.moduleActive )
   END_RUNG wire#w11
   // the same network as SCL:
   "EM02".PackML_Sts.Unit.sts_Completing_SC := ("EM02".PackML_Sts.Alarm.sts_Completing_SC OR NOT "EM02".PackML_Sts.Alarm.moduleActive) AND ("EM02".PackML_Sts.CM01.sts_Completing_SC OR NOT "EM02".PackML_Sts.CM01.moduleActive) AND ("EM02".PackML_Sts.CM02.sts_Completing_SC OR NOT "EM02".PackML_Sts.CM02.moduleActive) AND ("EM02".PackML_Sts.CM03.sts_Completing_SC OR NOT "EM02".PackML_Sts.CM03.moduleActive) AND ("EM02".PackML_Sts.CM04.sts_Completing_SC OR NOT "EM02".PackML_Sts.CM04.moduleActive) AND ("EM02".PackML_Sts.CM05.sts_Completing_SC OR NOT "EM02".PackML_Sts.CM05.moduleActive) AND ("EM02".PackML_Sts.CM06.sts_Completing_SC OR NOT "EM02".PackML_Sts.CM06.moduleActive) AND ("EM02".PackML_Sts.CM07.sts_Completing_SC OR NOT "EM02".PackML_Sts.CM07.moduleActive) AND ("EM02".PackML_Sts.CM08.sts_Completing_SC OR NOT "EM02".PackML_Sts.CM08.moduleActive) AND ("EM02".PackML_Sts.CM09.sts_Completing_SC OR NOT "EM02".PackML_Sts.CM09.moduleActive) AND ("EM02".PackML_Sts.CM10.sts_Completing_SC OR NOT "EM02".PackML_Sts.CM10.moduleActive);
END_REGION

REGION Network 21: Update the ENO Output value. (DO NOT REMOVE. Must be last rung)
   RUNG wire#powerrail
      ReturnCoil( TRUE )
   END_RUNG
   // the same network as SCL:
   ENO := TRUE;
   RETURN;
END_REGION
END_FUNCTION_BLOCK

ORGANIZATION_BLOCK "COMPLETE RESTART"   // OB100, LAD, Startup
TITLE = "Complete Restart"
{ S7_Optimized_Access := 'TRUE' }
VERSION : 0.1
// stored: AutoNumber true, IsIECCheckEnabled false, SetENOAutomatically false
   VAR_INPUT
      LostRetentive : Bool;   // True if retentive data are lost
      LostRTC : Bool;   // True if date and time are lost
   END_VAR
BEGIN
END_ORGANIZATION_BLOCK

ORGANIZATION_BLOCK "CYC_INT5"   // OB35, LAD, CyclicInterrupt
TITLE = "Cyclic Interrupt"
{ S7_Optimized_Access := 'TRUE' }
VERSION : 0.1
// stored: AutoNumber true, IsIECCheckEnabled false, SetENOAutomatically false
   VAR_INPUT
      Initial_Call : Bool;   // Initial call of this OB
      Event_Count : Int;   // Events discarded
   END_VAR
BEGIN
END_ORGANIZATION_BLOCK

ORGANIZATION_BLOCK "Programming error"   // OB121, LAD, ProgrammingError
{ S7_Optimized_Access := 'TRUE' }
VERSION : 0.1
// stored: IsIECCheckEnabled false, SetENOAutomatically false
   VAR_INPUT
      BlockNr : UInt;   // Number of causing block
      Reaction : USInt;   // 0:ignore, 1:substitute, 2:skip
      Fault_ID : Byte;   // Fault identifier
      BlockType : USInt;   // 16#01:OB, 16#02:FC, 16#03:FB, 16#04:SFC, 16#05:SFB, 16#06:DB: Type of block causing the error
      Area : USInt;   // Area where the error occured
      DBNr : DB_ANY;   // DB number if Area = DB or DI
      Csg_OBNr : OB_ANY;   // Number of OB causing the error
      Csg_Prio : USInt;   // Priority of OB causing the error
      Width : USInt;   // 0:bit, 1:byte, 2:word, 3:dword, 4:lword
   END_VAR
BEGIN
END_ORGANIZATION_BLOCK

ORGANIZATION_BLOCK "RACK_FLT"   // OB86, LAD, RackOrStationFailure
TITLE = "Loss Of Rack Fault"
{ S7_Optimized_Access := 'TRUE' }
VERSION : 0.1
// stored: IsIECCheckEnabled false, SetENOAutomatically false
   VAR_INPUT
      LADDR : HW_IO;   // Hardware identifier
      Event_Class : Byte;   // Event class
      Fault_ID : Byte;   // Fault identifier
   END_VAR
   VAR_TEMP
      OB86_RACKS_FLTD : Array[0..31] of Bool;
      OB86_DATE_TIME : Date_And_Time;   // Date and time OB86 started
   END_VAR
BEGIN
END_ORGANIZATION_BLOCK

ORGANIZATION_BLOCK "Time error interrupt"   // OB80, LAD, TimeErrorInterrupt
{ S7_Optimized_Access := 'TRUE' }
VERSION : 0.1
// stored: IsIECCheckEnabled false, SetENOAutomatically false
   VAR_INPUT
      Fault_ID : Byte;   // Fault identifier
      Csg_OBnr : OB_ANY;   // Number of OB causing the error
      Csg_Prio : UInt;   // Priority of OB causing the error
   END_VAR
BEGIN
END_ORGANIZATION_BLOCK

FUNCTION_BLOCK "EM00_CM06_Conveyor"   // FB2, LAD
TITLE = EM00_CM04
{ S7_Optimized_Access := 'TRUE' }
AUTHOR : tech.team.motioncontrol@siemens.com
FAMILY : CPG
VERSION : 1.1
// Support: tech.team.motioncontrol@siemens.com
// stored: AutoNumber true, IsIECCheckEnabled false, IsRetainMemResEnabled false, MemoryReserve 100, SetENOAutomatically false, UDAEnableTagReadback false
   VAR
      statDummyBool { ExternalAccessible := 'False'; ExternalVisible := 'False'; ExternalWritable := 'False'} : Bool;   // dummy bool - placeholder
   END_VAR
BEGIN

REGION Network 1: *** Begin the Setpoint Management Information Section ***
END_REGION

REGION Network 2: *** Begin the Logic Section ***
END_REGION

REGION Network 3: *** Begin the Event Information Section ***
END_REGION

REGION Network 4: *** Begin the State Model Status Feedback Section ***
END_REGION

REGION Network 5: *** Call the PackML Module Initialize Logic ***
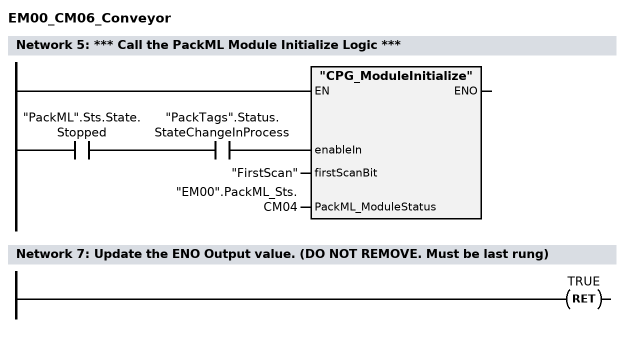
   RUNG wire#powerrail
      "CPG_ModuleInitialize"(enableIn := wire#w1, firstScanBit := "FirstScan", PackML_ModuleStatus := "EM00".PackML_Sts.CM04)
   END_RUNG
   RUNG wire#powerrail
      Contact( "PackML".Sts.State.Stopped )
      Contact( "PackTags".Status.StateChangeInProcess )
   END_RUNG wire#w1
   // the same network as SCL:
   "CPG_ModuleInitialize"(enableIn := "PackML".Sts.State.Stopped AND "PackTags".Status.StateChangeInProcess,
                          firstScanBit := "FirstScan",
                          PackML_ModuleStatus := "EM00".PackML_Sts.CM04);
END_REGION

REGION Network 7: Update the ENO Output value. (DO NOT REMOVE. Must be last rung)
   RUNG wire#powerrail
      ReturnCoil( TRUE )
   END_RUNG
   // the same network as SCL:
   ENO := TRUE;
   RETURN;
END_REGION
END_FUNCTION_BLOCK

FUNCTION_BLOCK "CPG_RecipeSetpoint_BOOL"
TITLE = CPG_RecipeSetpoint_BOOL
{ S7_Optimized_Access := 'TRUE' }
AUTHOR : 'tech.team.motioncontrol@siemens.com'
FAMILY : CPG
VERSION : 1.1
//Support: tech.team.motioncontrol@siemens.com
   VAR_INPUT 
      enable { ExternalAccessible := 'False'; ExternalVisible := 'False'; ExternalWritable := 'False'} : Bool;   // If true, setpoint changes are permitted
      disableRecipeControl { ExternalAccessible := 'False'; ExternalVisible := 'False'; ExternalWritable := 'False'} : Bool;   // If true, the setpoint is no longer handled as a recipe
   END_VAR

   VAR_OUTPUT 
      out { ExternalAccessible := 'False'; ExternalVisible := 'False'; ExternalWritable := 'False'} : Bool;   // Currently running recipe value
      changeEnabled { ExternalAccessible := 'False'; ExternalVisible := 'False'; ExternalWritable := 'False'} : Bool;   // Enable input is true, setpoint can be changed
      recipeControlDisabled { ExternalAccessible := 'False'; ExternalVisible := 'False'; ExternalWritable := 'False'} : Bool;   // The value is not subject to recipe controls
      changeNotAllowed { ExternalAccessible := 'False'; ExternalVisible := 'False'; ExternalWritable := 'False'} : Bool;   // Change is not permitted due to machine state
      recipeSetpointDifference { ExternalAccessible := 'False'; ExternalVisible := 'False'; ExternalWritable := 'False'} : Bool;   // The currently running (out) value and setpoint value are not equal
   END_VAR

   VAR_IN_OUT 
      recipeControl : "CPG_typeRecipeControl";   // Recipe control tag
      recipeSetpoint : "CPG_typeRecipeSetpoint_BOOL";   // Recipe setpoint tag
   END_VAR

   VAR 
      statFirstScan { ExternalAccessible := 'False'; ExternalVisible := 'False'; ExternalWritable := 'False'} : Bool := true;
      statPrevChangeNum { ExternalAccessible := 'False'; ExternalVisible := 'False'; ExternalWritable := 'False'} : Int;
      statPrevSaveNum { ExternalAccessible := 'False'; ExternalVisible := 'False'; ExternalWritable := 'False'} : Int;
      statPrevCopyNum { ExternalAccessible := 'False'; ExternalVisible := 'False'; ExternalWritable := 'False'} : Int;
      statPrevDeleteNum { ExternalAccessible := 'False'; ExternalVisible := 'False'; ExternalWritable := 'False'} : Int;
      statPrevOut { ExternalAccessible := 'False'; ExternalVisible := 'False'; ExternalWritable := 'False'} : Bool;
      statChangeNotAllowedTimer {InstructionName := 'TON_TIME'; LibVersion := '1.0'; ExternalAccessible := 'False'; ExternalVisible := 'False'; ExternalWritable := 'False'} : TON_TIME;
      statTimerEN { ExternalAccessible := 'False'; ExternalVisible := 'False'; ExternalWritable := 'False'} : Bool;
   END_VAR

   VAR CONSTANT 
      DELAY_TIME : Time := T#3s;
   END_VAR


BEGIN
	//============================================================================================================
	// SIEMENS AG
	// (c)Copyright 2019 All Rights Reserved
	//------------------------------------------------------------------------------------------------------------
	// Library: LCPG
	// Tested with: S7-1500 with FW version V2.1
	// Engineering: TIA Portal V14
	// Restrictions: ---
	// Requirements: S7-1500
	// Functionality: instantiate this once in the program for each recipe setpoint of BOOL
	// Support: tech.team.motioncontrol@siemens.com
	//------------------------------------------------------------------------------------------------------------
	// Change log table:
	// Version       Date               Expert in charge    Changes applied
	//  01.01.00     02.01.2019         KB                  Initial Release
	//============================================================================================================
	// Function : CPG_RecipeSetpoint_BOOL
	//============================================================================================================
	    
	// Language Selection
	#recipeSetpoint.CurrentName := #recipeSetpoint.SetpointName[#recipeControl.LanguageSelection];
	#recipeSetpoint.CurrentTextFalse := #recipeSetpoint.Text_False[#recipeControl.LanguageSelection];
	#recipeSetpoint.CurrentTextTrue := #recipeSetpoint.Text_True[#recipeControl.LanguageSelection];
	
	//Recipe Disable Control
	#recipeSetpoint.DisableRecipeControl := #disableRecipeControl;
	
	//Pass through enable bit
	#recipeSetpoint.SetpointChangeEnabled := #enable;
	
	//Set out value to match initial one on first scan
	IF #statFirstScan THEN
	    #recipeSetpoint.CurrentRecipeValue := #recipeSetpoint.RecipeValues[#recipeControl.CurrentRecipeID];
	    #recipeSetpoint.OUT := #recipeSetpoint.RecipeValues[#recipeControl.CurrentRecipeID];
	    #statFirstScan := false;
	END_IF;
	
	
	REGION RECIPE CONTROL
	    // Recipe Control - Change, Save, Copy, Delete, Revert setpoint, Save setpoint
	    IF NOT (#recipeSetpoint.DisableRecipeControl) THEN
	        //Recipe Change Command
	        IF #recipeControl.RecipeChangeNum <> #statPrevChangeNum THEN
	            #recipeSetpoint.OUT := #recipeSetpoint.RecipeValues[#recipeControl.CurrentRecipeID];
	            #statPrevChangeNum := #recipeControl.RecipeChangeNum;
	            // Prevents multiple commands from being executed if this instruction is not being scanned
	            #statPrevSaveNum := #recipeControl.RecipeSaveNum;
	            #statPrevCopyNum := #recipeControl.RecipeCopyNum;
	            #statPrevDeleteNum := #recipeControl.RecipeDeleteNum;
	        END_IF;
	        //Recipe Save Command
	        IF #recipeControl.RecipeSaveNum <> #statPrevSaveNum THEN
	            #recipeSetpoint.RecipeValues[#recipeControl.RecipeDestinationID] := #recipeSetpoint.OUT;
	            #statPrevSaveNum := #recipeControl.RecipeSaveNum;
	            // Prevents multiple commands from being executed if this instruction is not being scanned
	            #statPrevCopyNum := #recipeControl.RecipeCopyNum;
	            #statPrevDeleteNum := #recipeControl.RecipeDeleteNum;
	        END_IF;
	        //Recipe Copy Command
	        IF #recipeControl.RecipeCopyNum <> #statPrevCopyNum THEN
	            #recipeSetpoint.RecipeValues[#recipeControl.RecipeDestinationID] := #recipeSetpoint.RecipeValues[#recipeControl.RecipeSourceID];
	            #statPrevCopyNum := #recipeControl.RecipeCopyNum;
	            // Prevents multiple commands from being executed if this instruction is not being scanned
	            #statPrevDeleteNum := #recipeControl.RecipeDeleteNum;
	        END_IF;
	        //Recipe Delete Command
	        IF #recipeControl.RecipeDeleteNum <> #statPrevDeleteNum THEN
	            //edit this line to change the value a deleted recipe defaults to
	            #recipeSetpoint.RecipeValues[#recipeControl.RecipeDestinationID] := false;
	            #statPrevDeleteNum := #recipeControl.RecipeDeleteNum;
	        END_IF;
	        // Revert setpoint to saved value
	        IF #recipeSetpoint.RevertSetpoint THEN
	            #recipeSetpoint.OUT := #recipeSetpoint.RecipeValues[#recipeControl.CurrentRecipeID];
	        END_IF;
	        //Detect recipe/setpoint difference
	        IF (#recipeSetpoint.RecipeValues[#recipeControl.CurrentRecipeID] <> #recipeSetpoint.OUT) AND NOT (#recipeControl.RecipeChange) THEN
	            #recipeControl.RecipeSetpointDiff := true;  //signal to recipe control that a setpoint differs
	            #recipeSetpoint.RecipeSetpointDiff := true;
	        ELSE
	            #recipeSetpoint.RecipeSetpointDiff := false;
	        END_IF;
	        //Save setpoint
	        IF #recipeSetpoint.SaveSetpoint THEN
	            #recipeSetpoint.RecipeValues[#recipeControl.CurrentRecipeID] := #recipeSetpoint.OUT;
	        END_IF;
	        
	        //update values stored for current recipe & recipes A, B, & C
	        #recipeSetpoint.CurrentRecipeValue := #recipeSetpoint.RecipeValues[#recipeControl.CurrentRecipeID];
	        #recipeSetpoint.RecipeValueA := #recipeSetpoint.RecipeValues[#recipeControl.RecipeID_A];
	        #recipeSetpoint.RecipeValueB := #recipeSetpoint.RecipeValues[#recipeControl.RecipeID_B];
	        #recipeSetpoint.RecipeValueC := #recipeSetpoint.RecipeValues[#recipeControl.RecipeID_C];
	        
	    ELSE    //if recipe control is disabled, just update counters
	        #recipeSetpoint.RecipeSetpointDiff := false;
	        #statPrevChangeNum := #recipeControl.RecipeChangeNum;
	        #statPrevSaveNum := #recipeControl.RecipeSaveNum;
	        #statPrevCopyNum := #recipeControl.RecipeCopyNum;
	        #statPrevDeleteNum := #recipeControl.RecipeDeleteNum;
	    END_IF;
	END_REGION
	
	
	REGION UPDATE IN VALUE
	    //If ENABLE, then changes to the setpoint value are possible
	    //otherwise, updating the setpoint is not possible via changing RecipeSetpoint.IN
	    IF #enable THEN
	        //Clear status bit
	        #recipeSetpoint.SetpointChangeDisabled := false;
	        
	        // Check for input changed (due to user updating RecipeSetpoint.IN)
	        IF (#recipeSetpoint.IN XOR #recipeSetpoint.OUT) AND NOT (#recipeSetpoint.OUT XOR #statPrevOut) THEN
	            #recipeSetpoint.OUT := #recipeSetpoint.IN;
	        ELSE  // otherwise, update in to match out (this branch can execute due to a recipe change)
	            #recipeSetpoint.IN := #recipeSetpoint.OUT;
	        END_IF;
	        
	    ELSE
	        
	        // If in changes, revert and display message
	        IF (#recipeSetpoint.IN XOR #recipeSetpoint.OUT) OR #recipeSetpoint.RevertSetpoint THEN
	            #recipeSetpoint.IN := #recipeSetpoint.OUT;
	            #statTimerEN := false;
	            #recipeSetpoint.SetpointChangeDisabled := true;
	        END_IF;
	        
	        //display "setpoint changes not allowed" 3 seconds after inputting an invalid change
	        #statChangeNotAllowedTimer(IN := #statTimerEN,
	                               PT := #DELAY_TIME);
	        
	        // Continue to display the status bits for the duration of the timer.
	        IF #recipeSetpoint.SetpointChangeDisabled THEN
	            #statTimerEN := true;
	            #recipeSetpoint.SetpointChangeDisabled :=
	                #recipeSetpoint.SetpointChangeDisabled AND #statTimerEN AND NOT #statChangeNotAllowedTimer.Q;
	        END_IF;
	        
	    END_IF;
	END_REGION
	
	
	REGION DETERMINE HMI TEXTS
	    //This is a workaround because multiplexing inside a faceplate is not possible in V14SP1
	    IF #recipeSetpoint.OUT THEN
	        #recipeSetpoint.Out_Text := #recipeSetpoint.CurrentTextTrue;
	    ELSE
	        #recipeSetpoint.Out_Text := #recipeSetpoint.CurrentTextFalse;
	    END_IF;
	    IF #recipeSetpoint.CurrentRecipeValue THEN
	        #recipeSetpoint.CurrentRecipeValue_Text := #recipeSetpoint.CurrentTextTrue;
	    ELSE
	        #recipeSetpoint.CurrentRecipeValue_Text := #recipeSetpoint.CurrentTextFalse;
	    END_IF;
	    IF #recipeSetpoint.RecipeValueA THEN
	        #recipeSetpoint.RecipeA_Text := #recipeSetpoint.CurrentTextTrue;
	    ELSE
	        #recipeSetpoint.RecipeA_Text := #recipeSetpoint.CurrentTextFalse;
	    END_IF;
	    IF #recipeSetpoint.RecipeValueB THEN
	        #recipeSetpoint.RecipeB_Text := #recipeSetpoint.CurrentTextTrue;
	    ELSE
	        #recipeSetpoint.RecipeB_Text := #recipeSetpoint.CurrentTextFalse;
	    END_IF;
	    IF #recipeSetpoint.RecipeValueC THEN
	        #recipeSetpoint.RecipeC_Text := #recipeSetpoint.CurrentTextTrue;
	    ELSE
	        #recipeSetpoint.RecipeC_Text := #recipeSetpoint.CurrentTextFalse;
	    END_IF;
	END_REGION
	
	
	REGION SET OUTPUTS
	    #out := #recipeSetpoint.OUT;
	    #statPrevOut := #recipeSetpoint.OUT;
	    #changeNotAllowed := #recipeSetpoint.SetpointChangeDisabled;
	    #recipeSetpointDifference := #recipeSetpoint.RecipeSetpointDiff;
	    #recipeControlDisabled := #recipeSetpoint.DisableRecipeControl;
	    #changeEnabled := #recipeSetpoint.SetpointChangeEnabled;
	END_REGION
	
	
	//  -------------- END OF LOGIC -------------------------
	ENO := TRUE;   // Set the ENO output
END_FUNCTION_BLOCK

FUNCTION_BLOCK "CPG_RecipeSetpoint_DINT"
TITLE = CPG_RecipeSetpoint_DINT
{ S7_Optimized_Access := 'TRUE' }
AUTHOR : 'tech.team.motioncontrol@siemens.com'
FAMILY : CPG
VERSION : 1.1
//Support: tech.team.motioncontrol@siemens.com
   VAR_INPUT 
      enable { ExternalAccessible := 'False'; ExternalVisible := 'False'; ExternalWritable := 'False'} : Bool;   // If true, setpoint changes are permitted
      disableRecipeControl { ExternalAccessible := 'False'; ExternalVisible := 'False'; ExternalWritable := 'False'} : Bool;   // If true, the setpoint is no longer handled as a recipe
   END_VAR

   VAR_OUTPUT 
      out { ExternalAccessible := 'False'; ExternalVisible := 'False'; ExternalWritable := 'False'} : Real;   // Currently running recipe value
      changeEnabled { ExternalAccessible := 'False'; ExternalVisible := 'False'; ExternalWritable := 'False'} : Bool;   // Enable input is true, setpoint can be changed
      recipeControlDisabled { ExternalAccessible := 'False'; ExternalVisible := 'False'; ExternalWritable := 'False'} : Bool;   // The value is not subject to recipe controls
      changeNotAllowed { ExternalAccessible := 'False'; ExternalVisible := 'False'; ExternalWritable := 'False'} : Bool;   // Change is not permitted due to machine state
      recipeSetpointDifference { ExternalAccessible := 'False'; ExternalVisible := 'False'; ExternalWritable := 'False'} : Bool;   // The currently running (out) value and setpoint value are not equal
      minLimitExceeded { ExternalAccessible := 'False'; ExternalVisible := 'False'; ExternalWritable := 'False'} : Bool;   // Minimum limit exceeded
      maxLimitExceeded { ExternalAccessible := 'False'; ExternalVisible := 'False'; ExternalWritable := 'False'} : Bool;   // Maximum limit exceeded
   END_VAR

   VAR_IN_OUT 
      recipeControl : "CPG_typeRecipeControl";   // Recipe control tag
      recipeSetpoint : "CPG_typeRecipeSetpoint_DINT";   // Recipe setpoint tag
   END_VAR

   VAR 
      statFirstScan { ExternalAccessible := 'False'; ExternalVisible := 'False'; ExternalWritable := 'False'} : Bool := true;
      statPrevChangeNum { ExternalAccessible := 'False'; ExternalVisible := 'False'; ExternalWritable := 'False'} : Int;
      statPrevSaveNum { ExternalAccessible := 'False'; ExternalVisible := 'False'; ExternalWritable := 'False'} : Int;
      statPrevCopyNum { ExternalAccessible := 'False'; ExternalVisible := 'False'; ExternalWritable := 'False'} : Int;
      statPrevDeleteNum { ExternalAccessible := 'False'; ExternalVisible := 'False'; ExternalWritable := 'False'} : Int;
      statPrevOut { ExternalAccessible := 'False'; ExternalVisible := 'False'; ExternalWritable := 'False'} : DInt;
      statLimitsTimer {InstructionName := 'TP_TIME'; LibVersion := '1.0'; ExternalAccessible := 'False'; ExternalVisible := 'False'; ExternalWritable := 'False'} : TP_TIME;
      statLimitsTimerEN { ExternalAccessible := 'False'; ExternalVisible := 'False'; ExternalWritable := 'False'} : Bool;
      statChangeNotAllowedTimer {InstructionName := 'TON_TIME'; LibVersion := '1.0'; ExternalAccessible := 'False'; ExternalVisible := 'False'; ExternalWritable := 'False'} : TON_TIME;
      statTimerEN { ExternalAccessible := 'False'; ExternalVisible := 'False'; ExternalWritable := 'False'} : Bool;
   END_VAR

   VAR_TEMP 
      tempLimit : DInt;
   END_VAR

   VAR CONSTANT 
      DELAY_TIME : Time := T#3s;
   END_VAR


BEGIN
	//============================================================================================================
	// SIEMENS AG
	// (c)Copyright 2019 All Rights Reserved
	//------------------------------------------------------------------------------------------------------------
	// Library: LCPG
	// Tested with: S7-1500 with FW version V2.1
	// Engineering: TIA Portal V14
	// Restrictions: ---
	// Requirements: S7-1500
	// Functionality: instantiate this once in the program for each recipe setpoint of DINT
	// Support: tech.team.motioncontrol@siemens.com
	//------------------------------------------------------------------------------------------------------------
	// Change log table:
	// Version       Date               Expert in charge    Changes applied
	//  01.01.00     02.01.2019         KB                  Initial Release
	//============================================================================================================
	// Function : CPG_RecipeSetpoint_DINT
	//============================================================================================================
	
	// Language Selection
	#recipeSetpoint.CurrentName := #recipeSetpoint.SetpointName[#recipeControl.LanguageSelection];
	
	//Recipe Disable Control
	#recipeSetpoint.DisableRecipeControl := #disableRecipeControl;
	
	//Pass through enable bit
	#recipeSetpoint.SetpointChangeEnabled := #enable;
	
	//Set out value to match initial one on first scan
	IF #statFirstScan THEN
	    #recipeSetpoint.CurrentRecipeValue := #recipeSetpoint.RecipeValues[#recipeControl.CurrentRecipeID];
	    #recipeSetpoint.OUT := #recipeSetpoint.RecipeValues[#recipeControl.CurrentRecipeID];
	    #statFirstScan := false;
	END_IF;
	
	
	REGION CHECK LIMITS
	    //checks if min & max limits are valid.  If they are not in order, swap them
	    IF #recipeSetpoint.minLimit > #recipeSetpoint.maxLimit THEN
	        #tempLimit := #recipeSetpoint.minLimit;
	        #recipeSetpoint.minLimit := #recipeSetpoint.maxLimit;
	        #recipeSetpoint.maxLimit := #tempLimit;
	    END_IF;
	    
	    //checks if the saved recipe value is outside the bounds, either due to a runtime change of the limits or a bad configuration
	    //if problems, and recipe control is on, set the saved value to the default (min limit, same as recipeDelete)
	    //Note that this check is only on the current recipe, and also is only performed if recipeControlDisable is false
	    IF #recipeSetpoint.RecipeValues[#recipeControl.CurrentRecipeID] < #recipeSetpoint.minLimit
	        OR #recipeSetpoint.RecipeValues[#recipeControl.CurrentRecipeID] > #recipeSetpoint.maxLimit
	        AND NOT (#recipeSetpoint.DisableRecipeControl) THEN
	        #recipeSetpoint.RecipeValues[#recipeControl.CurrentRecipeID] := #recipeSetpoint.minLimit;
	    END_IF;
	    
	    //Checks the out value.  Note that this value matters even if recipeControlDisable is true
	    //If the value is a being controlled, then set the value to the (guarenteed to be in range) saved recipe value
	    //If the value is not being treated as a recipe, set it to the default (minlimit)
	    IF #recipeSetpoint.OUT < #recipeSetpoint.minLimit OR #recipeSetpoint.OUT > #recipeSetpoint.maxLimit THEN
	        IF NOT (#recipeSetpoint.DisableRecipeControl) THEN
	            #recipeSetpoint.OUT := #recipeSetpoint.RecipeValues[#recipeControl.CurrentRecipeID];
	        ELSE
	            #recipeSetpoint.OUT := #recipeSetpoint.minLimit;
	        END_IF;
	    END_IF;
	END_REGION
	
	
	REGION RECIPE CONTROL
	    // Recipe Control - Change, Save, Copy, Delete, Revert setpoint, Save setpoint
	    IF NOT (#recipeSetpoint.DisableRecipeControl) THEN
	        //Recipe Change Command
	        IF #recipeControl.RecipeChangeNum <> #statPrevChangeNum THEN
	            #recipeSetpoint.OUT := #recipeSetpoint.RecipeValues[#recipeControl.CurrentRecipeID];
	            #statPrevChangeNum := #recipeControl.RecipeChangeNum;
	            // Prevents multiple commands from being executed if this instruction is not being scanned
	            #statPrevSaveNum := #recipeControl.RecipeSaveNum;
	            #statPrevCopyNum := #recipeControl.RecipeCopyNum;
	            #statPrevDeleteNum := #recipeControl.RecipeDeleteNum;
	        END_IF;
	        //Recipe Save Command
	        IF #recipeControl.RecipeSaveNum <> #statPrevSaveNum THEN
	            #recipeSetpoint.RecipeValues[#recipeControl.RecipeDestinationID] := #recipeSetpoint.OUT;
	            #statPrevSaveNum := #recipeControl.RecipeSaveNum;
	            // Prevents multiple commands from being executed if this instruction is not being scanned
	            #statPrevCopyNum := #recipeControl.RecipeCopyNum;
	            #statPrevDeleteNum := #recipeControl.RecipeDeleteNum;
	        END_IF;
	        //Recipe Copy Command
	        IF #recipeControl.RecipeCopyNum <> #statPrevCopyNum THEN
	            #recipeSetpoint.RecipeValues[#recipeControl.RecipeDestinationID] := #recipeSetpoint.RecipeValues[#recipeControl.RecipeSourceID];
	            #statPrevCopyNum := #recipeControl.RecipeCopyNum;
	            // Prevents multiple commands from being executed if this instruction is not being scanned
	            #statPrevDeleteNum := #recipeControl.RecipeDeleteNum;
	        END_IF;
	        //Recipe Delete Command
	        IF #recipeControl.RecipeDeleteNum <> #statPrevDeleteNum THEN
	            //edit this line to change the value a deleted recipe defaults to
	            #recipeSetpoint.RecipeValues[#recipeControl.RecipeDestinationID] := #recipeSetpoint.minLimit;
	            #statPrevDeleteNum := #recipeControl.RecipeDeleteNum;
	        END_IF;
	        // Revert setpoint to saved value
	        IF #recipeSetpoint.RevertSetpoint THEN
	            #recipeSetpoint.OUT := #recipeSetpoint.RecipeValues[#recipeControl.CurrentRecipeID];
	        END_IF;
	        //Detect recipe/setpoint difference
	        IF (#recipeSetpoint.RecipeValues[#recipeControl.CurrentRecipeID] <> #recipeSetpoint.OUT) AND NOT (#recipeControl.RecipeChange) THEN
	            #recipeControl.RecipeSetpointDiff := true;  //signal to recipe control that a setpoint differs
	            #recipeSetpoint.RecipeSetpointDiff := true;
	        ELSE
	            #recipeSetpoint.RecipeSetpointDiff := false;
	        END_IF;
	        //Save setpoint
	        IF #recipeSetpoint.SaveSetpoint THEN
	            #recipeSetpoint.RecipeValues[#recipeControl.CurrentRecipeID] := #recipeSetpoint.OUT;
	        END_IF;
	        
	        //update values stored for current recipe & recipes A, B, & C
	        #recipeSetpoint.CurrentRecipeValue := #recipeSetpoint.RecipeValues[#recipeControl.CurrentRecipeID];
	        #recipeSetpoint.RecipeValueA := #recipeSetpoint.RecipeValues[#recipeControl.RecipeID_A];
	        #recipeSetpoint.RecipeValueB := #recipeSetpoint.RecipeValues[#recipeControl.RecipeID_B];
	        #recipeSetpoint.RecipeValueC := #recipeSetpoint.RecipeValues[#recipeControl.RecipeID_C];
	        
	    ELSE    //if recipe control is disabled, just update counters
	        #recipeSetpoint.RecipeSetpointDiff := false;
	        #statPrevChangeNum := #recipeControl.RecipeChangeNum;
	        #statPrevSaveNum := #recipeControl.RecipeSaveNum;
	        #statPrevCopyNum := #recipeControl.RecipeCopyNum;
	        #statPrevDeleteNum := #recipeControl.RecipeDeleteNum;
	    END_IF;
	END_REGION
	
	REGION UPDATE IN VALUE
	    //If ENABLE, then changes to the setpoint value are possible
	    //otherwise, updating the setpoint is not possible via changing RecipeSetpoint.IN
	    IF #enable THEN
	        //Clear status bit
	        #recipeSetpoint.SetpointChangeDisabled := false;
	        
	        // Check for value within limits and input changed (due to user updating RecipeSetpoint.IN)
	        IF (#recipeSetpoint.minLimit <= #recipeSetpoint.IN) AND (#recipeSetpoint.IN <= #recipeSetpoint.maxLimit) AND
	            (#recipeSetpoint.IN <> #recipeSetpoint.OUT) AND (#recipeSetpoint.OUT = #statPrevOut) THEN
	            #recipeSetpoint.OUT := #recipeSetpoint.IN;
	            #recipeSetpoint.minLimitReached := false;
	            #recipeSetpoint.maxLimitReached := false;
	        // Check for value within limits and output changed (due to a recipe change)
	        ELSIF (#recipeSetpoint.minLimit <= #recipeSetpoint.IN) AND (#recipeSetpoint.IN <= #recipeSetpoint.maxLimit) AND
	            (#recipeSetpoint.IN <> #recipeSetpoint.OUT) AND (#recipeSetpoint.OUT <> #statPrevOut) THEN
	            #recipeSetpoint.IN := #recipeSetpoint.OUT;
	            #recipeSetpoint.minLimitReached := false;
	            #recipeSetpoint.maxLimitReached := false;
	        // Check for value below minimum limit
	        ELSIF (#recipeSetpoint.minLimit > #recipeSetpoint.IN) THEN
	            #statLimitsTimerEN := true;
	            #recipeSetpoint.IN := #recipeSetpoint.OUT;
	            #recipeSetpoint.minLimitReached := true;
	            #recipeSetpoint.maxLimitReached := false;
	        // Check for value above maximum limit
	        ELSIF (#recipeSetpoint.maxLimit < #recipeSetpoint.IN) THEN
	            #statLimitsTimerEN := true;
	            #recipeSetpoint.IN := #recipeSetpoint.OUT;
	            #recipeSetpoint.minLimitReached := false;
	            #recipeSetpoint.maxLimitReached := true;
	        END_IF;
	        
	        #statLimitsTimer(IN := #statLimitsTimerEN,
	                     PT := #DELAY_TIME);
	        
	        // Continue to display the status bits for the duration of the timer.
	        IF #recipeSetpoint.minLimitReached OR #recipeSetpoint.maxLimitReached THEN
	            #statLimitsTimerEN := false;
	            #recipeSetpoint.minLimitReached := #recipeSetpoint.minLimitReached AND #statLimitsTimer.Q;
	            #recipeSetpoint.maxLimitReached := #recipeSetpoint.maxLimitReached AND #statLimitsTimer.Q;
	        END_IF;
	        
	    ELSE
	        
	        // If IN changes, revert and display message
	        IF (#recipeSetpoint.IN <> #recipeSetpoint.OUT) OR #recipeSetpoint.RevertSetpoint THEN
	            #recipeSetpoint.IN := #recipeSetpoint.OUT;
	            #statTimerEN := false;
	            #recipeSetpoint.SetpointChangeDisabled := true;
	            #recipeSetpoint.minLimitReached := false;
	            #recipeSetpoint.maxLimitReached := false;
	        END_IF;
	        
	        //display "setpoint changes not allowed" 3 seconds after inputting an invalid change
	        #statChangeNotAllowedTimer(IN := #statTimerEN,
	                               PT := #DELAY_TIME);
	        
	        // Continue to display the status bits for the duration of the timer.
	        IF #recipeSetpoint.SetpointChangeDisabled THEN
	            #statTimerEN := true;
	            #recipeSetpoint.SetpointChangeDisabled :=
	                #recipeSetpoint.SetpointChangeDisabled AND #statTimerEN AND NOT #statChangeNotAllowedTimer.Q;
	        END_IF;
	        
	    END_IF;
	END_REGION
	
	
	REGION SET OUTPUTS
	    #out := #recipeSetpoint.OUT;
	    #statPrevOut := #recipeSetpoint.OUT;
	    #changeNotAllowed := #recipeSetpoint.SetpointChangeDisabled;
	    #recipeSetpointDifference := #recipeSetpoint.RecipeSetpointDiff;
	    #recipeControlDisabled := #recipeSetpoint.DisableRecipeControl;
	    #changeEnabled := #recipeSetpoint.SetpointChangeEnabled;
	    #minLimitExceeded := #recipeSetpoint.minLimitReached;
	    #maxLimitExceeded := #recipeSetpoint.maxLimitReached;
	END_REGION
	
	//  -------------- END OF LOGIC -------------------------
	ENO := TRUE;   // Set the ENO output
END_FUNCTION_BLOCK

FUNCTION_BLOCK "CPG_RecipeSetpoint_REAL"
TITLE = CPG_RecipeSetpoint_REAL
{ S7_Optimized_Access := 'TRUE' }
AUTHOR : 'tech.team.motioncontrol@siemens.com'
FAMILY : CPG
VERSION : 1.1
//Support: tech.team.motioncontrol@siemens.com
   VAR_INPUT 
      enable { ExternalAccessible := 'False'; ExternalVisible := 'False'; ExternalWritable := 'False'} : Bool;   // If true, setpoint changes are permitted
      disableRecipeControl { ExternalAccessible := 'False'; ExternalVisible := 'False'; ExternalWritable := 'False'; S7_HiddenAssignment := 'HideIfNoParamAssigned'} : Bool;   // If true, the setpoint is no longer handled as a recipe
   END_VAR

   VAR_OUTPUT 
      out { ExternalAccessible := 'False'; ExternalVisible := 'False'; ExternalWritable := 'False'} : Real;   // Currently running recipe value
      changeEnabled { ExternalAccessible := 'False'; ExternalVisible := 'False'; ExternalWritable := 'False'} : Bool;   // Enable input is true, setpoint can be changed
      recipeControlDisabled { ExternalAccessible := 'False'; ExternalVisible := 'False'; ExternalWritable := 'False'} : Bool;   // The value is not subject to recipe controls
      changeNotAllowed { ExternalAccessible := 'False'; ExternalVisible := 'False'; ExternalWritable := 'False'} : Bool;   // Change is not permitted due to machine state
      recipeSetpointDifference { ExternalAccessible := 'False'; ExternalVisible := 'False'; ExternalWritable := 'False'} : Bool;   // The currently running (out) value and setpoint value are not equal
      minLimitExceeded { ExternalAccessible := 'False'; ExternalVisible := 'False'; ExternalWritable := 'False'} : Bool;   // Minimum limit exceeded
      maxLimitExceeded { ExternalAccessible := 'False'; ExternalVisible := 'False'; ExternalWritable := 'False'} : Bool;   // Maximum limit exceeded
   END_VAR

   VAR_IN_OUT 
      recipeControl : "CPG_typeRecipeControl";   // Recipe control tag
      recipeSetpoint : "CPG_typeRecipeSetpoint_REAL";   // Recipe setpoint tag
   END_VAR

   VAR 
      statFirstScan { ExternalAccessible := 'False'; ExternalVisible := 'False'; ExternalWritable := 'False'} : Bool := true;
      statPrevChangeNum { ExternalAccessible := 'False'; ExternalVisible := 'False'; ExternalWritable := 'False'} : Int;
      statPrevSaveNum { ExternalAccessible := 'False'; ExternalVisible := 'False'; ExternalWritable := 'False'} : Int;
      statPrevCopyNum { ExternalAccessible := 'False'; ExternalVisible := 'False'; ExternalWritable := 'False'} : Int;
      statPrevDeleteNum { ExternalAccessible := 'False'; ExternalVisible := 'False'; ExternalWritable := 'False'} : Int;
      statPrevOut { ExternalAccessible := 'False'; ExternalVisible := 'False'; ExternalWritable := 'False'} : Real;
      statLimitsTimer {InstructionName := 'TP_TIME'; LibVersion := '1.0'; ExternalAccessible := 'False'; ExternalVisible := 'False'; ExternalWritable := 'False'} : TP_TIME;
      statLimitsTimerEN { ExternalAccessible := 'False'; ExternalVisible := 'False'; ExternalWritable := 'False'} : Bool;
      statChangeNotAllowedTimer {InstructionName := 'TON_TIME'; LibVersion := '1.0'; ExternalAccessible := 'False'; ExternalVisible := 'False'; ExternalWritable := 'False'} : TON_TIME;
      statTimerEN { ExternalAccessible := 'False'; ExternalVisible := 'False'; ExternalWritable := 'False'} : Bool;
   END_VAR

   VAR_TEMP 
      tempLimit : Real;
   END_VAR

   VAR CONSTANT 
      DELAY_TIME : Time := T#3s;
   END_VAR


BEGIN
	//============================================================================================================
	// SIEMENS AG
	// (c)Copyright 2019 All Rights Reserved
	//------------------------------------------------------------------------------------------------------------
	// Library: LCPG
	// Tested with: S7-1500 with FW version V2.1
	// Engineering: TIA Portal V14
	// Restrictions: ---
	// Requirements: S7-1500
	// Functionality: instantiate this once in the program for each recipe setpoint of REAL
	// Support: tech.team.motioncontrol@siemens.com
	//------------------------------------------------------------------------------------------------------------
	// Change log table:
	// Version       Date               Expert in charge    Changes applied
	//  01.01.00     02.01.2019         KB                  Initial Release
	//============================================================================================================
	// Function : CPG_RecipeSetpoint_REAL
	//============================================================================================================
	
	// Language Selection
	#recipeSetpoint.CurrentName := #recipeSetpoint.SetpointName[#recipeControl.LanguageSelection];
	
	//Recipe Disable Control
	#recipeSetpoint.DisableRecipeControl := #disableRecipeControl;
	
	//Pass through enable bit
	#recipeSetpoint.SetpointChangeEnabled := #enable;
	
	//Set out value to match initial one on first scan
	IF #statFirstScan THEN
	    #recipeSetpoint.CurrentRecipeValue := #recipeSetpoint.RecipeValues[#recipeControl.CurrentRecipeID];
	    #recipeSetpoint.OUT := #recipeSetpoint.RecipeValues[#recipeControl.CurrentRecipeID];
	    #statFirstScan := false;
	END_IF;
	
	
	REGION CHECK LIMITS
	    //checks if min & max limits are valid.  If they are not in order, swap them
	    IF #recipeSetpoint.minLimit > #recipeSetpoint.maxLimit THEN
	        #tempLimit := #recipeSetpoint.minLimit;
	        #recipeSetpoint.minLimit := #recipeSetpoint.maxLimit;
	        #recipeSetpoint.maxLimit := #tempLimit;
	    END_IF;
	    
	    //checks if the saved recipe value is outside the bounds, either due to a runtime change of the limits or a bad configuration
	    //if problems, and recipe control is on, set the saved value to the default (min limit, same as recipeDelete)
	    //Note that this check is only on the current recipe, and also is only performed if recipeControlDisable is false
	    IF #recipeSetpoint.RecipeValues[#recipeControl.CurrentRecipeID] < #recipeSetpoint.minLimit
	        OR #recipeSetpoint.RecipeValues[#recipeControl.CurrentRecipeID] > #recipeSetpoint.maxLimit
	        AND NOT (#recipeSetpoint.DisableRecipeControl) THEN
	        #recipeSetpoint.RecipeValues[#recipeControl.CurrentRecipeID] := #recipeSetpoint.minLimit;
	    END_IF;
	    
	    //Checks the out value.  Note that this value matters even if recipeControlDisable is true
	    //If the value is a being controlled, then set the value to the (guarenteed to be in range) saved recipe value
	    //If the value is not being treated as a recipe, set it to the default (minlimit)
	    IF #recipeSetpoint.OUT < #recipeSetpoint.minLimit OR #recipeSetpoint.OUT > #recipeSetpoint.maxLimit THEN
	        IF NOT (#recipeSetpoint.DisableRecipeControl) THEN
	            #recipeSetpoint.OUT := #recipeSetpoint.RecipeValues[#recipeControl.CurrentRecipeID];
	        ELSE
	            #recipeSetpoint.OUT := #recipeSetpoint.minLimit;
	        END_IF;
	    END_IF;
	END_REGION
	
	
	REGION RECIPE CONTROL
	    // Recipe Control - Change, Save, Copy, Delete, Revert setpoint, Save setpoint
	    IF NOT (#recipeSetpoint.DisableRecipeControl) THEN
	        //Recipe Change Command
	        IF #recipeControl.RecipeChangeNum <> #statPrevChangeNum THEN
	            #recipeSetpoint.OUT := #recipeSetpoint.RecipeValues[#recipeControl.CurrentRecipeID];
	            #statPrevChangeNum := #recipeControl.RecipeChangeNum;
	            // Prevents multiple commands from being executed if this instruction is not being scanned
	            #statPrevSaveNum := #recipeControl.RecipeSaveNum;
	            #statPrevCopyNum := #recipeControl.RecipeCopyNum;
	            #statPrevDeleteNum := #recipeControl.RecipeDeleteNum;
	        END_IF;
	        //Recipe Save Command
	        IF #recipeControl.RecipeSaveNum <> #statPrevSaveNum THEN
	            #recipeSetpoint.RecipeValues[#recipeControl.RecipeDestinationID] := #recipeSetpoint.OUT;
	            #statPrevSaveNum := #recipeControl.RecipeSaveNum;
	            // Prevents multiple commands from being executed if this instruction is not being scanned
	            #statPrevCopyNum := #recipeControl.RecipeCopyNum;
	            #statPrevDeleteNum := #recipeControl.RecipeDeleteNum;
	        END_IF;
	        //Recipe Copy Command
	        IF #recipeControl.RecipeCopyNum <> #statPrevCopyNum THEN
	            #recipeSetpoint.RecipeValues[#recipeControl.RecipeDestinationID] := #recipeSetpoint.RecipeValues[#recipeControl.RecipeSourceID];
	            #statPrevCopyNum := #recipeControl.RecipeCopyNum;
	            // Prevents multiple commands from being executed if this instruction is not being scanned
	            #statPrevDeleteNum := #recipeControl.RecipeDeleteNum;
	        END_IF;
	        //Recipe Delete Command
	        IF #recipeControl.RecipeDeleteNum <> #statPrevDeleteNum THEN
	            //edit this line to change the value a deleted recipe defaults to
	            #recipeSetpoint.RecipeValues[#recipeControl.RecipeDestinationID] := #recipeSetpoint.minLimit;   
	            #statPrevDeleteNum := #recipeControl.RecipeDeleteNum;
	        END_IF;
	        // Revert setpoint to saved value
	        IF #recipeSetpoint.RevertSetpoint THEN
	            #recipeSetpoint.OUT := #recipeSetpoint.RecipeValues[#recipeControl.CurrentRecipeID];
	        END_IF;
	        //Detect recipe/setpoint difference
	        IF (#recipeSetpoint.RecipeValues[#recipeControl.CurrentRecipeID] <> #recipeSetpoint.OUT) AND NOT (#recipeControl.RecipeChange) THEN
	            #recipeControl.RecipeSetpointDiff := true;  //signal to recipe control that a setpoint differs
	            #recipeSetpoint.RecipeSetpointDiff := true;
	        ELSE
	            #recipeSetpoint.RecipeSetpointDiff := false;
	        END_IF;
	        //Save setpoint
	        IF #recipeSetpoint.SaveSetpoint THEN
	            #recipeSetpoint.RecipeValues[#recipeControl.CurrentRecipeID] := #recipeSetpoint.OUT;
	        END_IF;
	        
	        
	        //update values stored for current recipe & recipes A, B, & C
	        #recipeSetpoint.CurrentRecipeValue := #recipeSetpoint.RecipeValues[#recipeControl.CurrentRecipeID];
	        #recipeSetpoint.RecipeValueA := #recipeSetpoint.RecipeValues[#recipeControl.RecipeID_A];
	        #recipeSetpoint.RecipeValueB := #recipeSetpoint.RecipeValues[#recipeControl.RecipeID_B];
	        #recipeSetpoint.RecipeValueC := #recipeSetpoint.RecipeValues[#recipeControl.RecipeID_C];
	        
	    ELSE    //if recipe control is disabled, just update counters
	        #recipeSetpoint.RecipeSetpointDiff := false;
	        #statPrevChangeNum := #recipeControl.RecipeChangeNum;
	        #statPrevSaveNum := #recipeControl.RecipeSaveNum;
	        #statPrevCopyNum := #recipeControl.RecipeCopyNum;
	        #statPrevDeleteNum := #recipeControl.RecipeDeleteNum;
	    END_IF;
	END_REGION
	
	
	REGION UPDATE IN VALUE
	    //If ENABLE, then changes to the setpoint value are possible
	    //otherwise, updating the setpoint is not possible via changing RecipeSetpoint.IN
	    IF #enable THEN
	        //Clear status bit
	        #recipeSetpoint.SetpointChangeDisabled := false;
	        
	        // Check for value within limits and input changed (due to user updating RecipeSetpoint.IN)
	        IF (#recipeSetpoint.minLimit <= #recipeSetpoint.IN) AND (#recipeSetpoint.IN <= #recipeSetpoint.maxLimit) AND
	            (#recipeSetpoint.IN <> #recipeSetpoint.OUT) AND (#recipeSetpoint.OUT = #statPrevOut) THEN
	            #recipeSetpoint.OUT := #recipeSetpoint.IN;
	            #recipeSetpoint.minLimitReached := false;
	            #recipeSetpoint.maxLimitReached := false;
	        // Check for value within limits and output changed (due to a recipe change)
	        ELSIF (#recipeSetpoint.minLimit <= #recipeSetpoint.IN) AND (#recipeSetpoint.IN <= #recipeSetpoint.maxLimit) AND
	            (#recipeSetpoint.IN <> #recipeSetpoint.OUT) AND (#recipeSetpoint.OUT <> #statPrevOut) THEN
	            #recipeSetpoint.IN := #recipeSetpoint.OUT;
	            #recipeSetpoint.minLimitReached := false;
	            #recipeSetpoint.maxLimitReached := false;
	        // Check for value below minimum limit
	        ELSIF (#recipeSetpoint.minLimit > #recipeSetpoint.IN) THEN
	            #statLimitsTimerEN := true;
	            #recipeSetpoint.IN := #recipeSetpoint.OUT;
	            #recipeSetpoint.minLimitReached := true;
	            #recipeSetpoint.maxLimitReached := false;
	        // Check for value above maximum limit
	        ELSIF (#recipeSetpoint.maxLimit < #recipeSetpoint.IN) THEN
	            #statLimitsTimerEN := true;
	            #recipeSetpoint.IN := #recipeSetpoint.OUT;
	            #recipeSetpoint.minLimitReached := false;
	            #recipeSetpoint.maxLimitReached := true;
	        END_IF;
	        
	        #statLimitsTimer(IN := #statLimitsTimerEN,
	                     PT := #DELAY_TIME);
	        
	        // Continue to display the status bits for the duration of the timer.
	        IF #recipeSetpoint.minLimitReached OR #recipeSetpoint.maxLimitReached THEN
	            #statLimitsTimerEN := false;
	            #recipeSetpoint.minLimitReached := #recipeSetpoint.minLimitReached AND #statLimitsTimer.Q;
	            #recipeSetpoint.maxLimitReached := #recipeSetpoint.maxLimitReached AND #statLimitsTimer.Q;
	        END_IF;
	        
	    ELSE
	        
	        // If IN changes, revert and display message
	        IF (#recipeSetpoint.IN <> #recipeSetpoint.OUT) OR #recipeSetpoint.RevertSetpoint THEN
	            #recipeSetpoint.IN := #recipeSetpoint.OUT;
	            #statTimerEN := false;
	            #recipeSetpoint.SetpointChangeDisabled := true;
	            #recipeSetpoint.minLimitReached := false;
	            #recipeSetpoint.maxLimitReached := false;
	        END_IF;
	        
	        //display "setpoint changes not allowed" 3 seconds after inputting an invalid change
	        #statChangeNotAllowedTimer(IN := #statTimerEN,
	                               PT := #DELAY_TIME);
	        
	        // Continue to display the status bits for the duration of the timer.
	        IF #recipeSetpoint.SetpointChangeDisabled THEN
	            #statTimerEN := true;
	            #recipeSetpoint.SetpointChangeDisabled :=
	                #recipeSetpoint.SetpointChangeDisabled AND #statTimerEN AND NOT #statChangeNotAllowedTimer.Q;
	        END_IF;
	        
	    END_IF;
	END_REGION
	
	
	REGION SET OUTPUTS
	    #out := #recipeSetpoint.OUT;
	    #statPrevOut := #recipeSetpoint.OUT;
	    #changeNotAllowed := #recipeSetpoint.SetpointChangeDisabled;
	    #recipeSetpointDifference := #recipeSetpoint.RecipeSetpointDiff;
	    #recipeControlDisabled := #recipeSetpoint.DisableRecipeControl;
	    #changeEnabled := #recipeSetpoint.SetpointChangeEnabled;
	    #minLimitExceeded := #recipeSetpoint.minLimitReached;
	    #maxLimitExceeded := #recipeSetpoint.maxLimitReached;
	END_REGION
	
	//  -------------- END OF LOGIC -------------------------
	ENO := TRUE;   // Set the ENO output
END_FUNCTION_BLOCK

FUNCTION_BLOCK "CPG_RecipeSetpoint_STRING"
TITLE = CPG_RecipeSetpoint_STRING
{ S7_Optimized_Access := 'TRUE' }
AUTHOR : 'tech.team.motioncontrol@siemens.com'
FAMILY : CPG
VERSION : 1.1
//Support: tech.team.motioncontrol@siemens.com
   VAR_INPUT 
      enable { ExternalAccessible := 'False'; ExternalVisible := 'False'; ExternalWritable := 'False'} : Bool;   // If true, setpoint changes are permitted
      disableRecipeControl { ExternalAccessible := 'False'; ExternalVisible := 'False'; ExternalWritable := 'False'} : Bool;   // If true, the setpoint is no longer handled as a recipe
   END_VAR

   VAR_OUTPUT 
      out { ExternalAccessible := 'False'; ExternalVisible := 'False'; ExternalWritable := 'False'} : String[60];   // Currently running recipe value
      changeEnabled { ExternalAccessible := 'False'; ExternalVisible := 'False'; ExternalWritable := 'False'} : Bool;   // Enable input is true, setpoint can be changed
      recipeControlDisabled { ExternalAccessible := 'False'; ExternalVisible := 'False'; ExternalWritable := 'False'} : Bool;   // The value is not subject to recipe controls
      changeNotAllowed { ExternalAccessible := 'False'; ExternalVisible := 'False'; ExternalWritable := 'False'} : Bool;   // Change is not permitted due to machine state
      recipeSetpointDifference { ExternalAccessible := 'False'; ExternalVisible := 'False'; ExternalWritable := 'False'} : Bool;   // The currently running (out) value and setpoint value are not equal
   END_VAR

   VAR_IN_OUT 
      recipeControl : "CPG_typeRecipeControl";   // Recipe control tag
      recipeSetpoint : "CPG_typeRecipeSetpoint_STRING";   // Recipe setpoint tag
   END_VAR

   VAR 
      statFirstScan { ExternalAccessible := 'False'; ExternalVisible := 'False'; ExternalWritable := 'False'} : Bool := true;
      statPrevChangeNum { ExternalAccessible := 'False'; ExternalVisible := 'False'; ExternalWritable := 'False'} : Int;
      statPrevSaveNum { ExternalAccessible := 'False'; ExternalVisible := 'False'; ExternalWritable := 'False'} : Int;
      statPrevCopyNum { ExternalAccessible := 'False'; ExternalVisible := 'False'; ExternalWritable := 'False'} : Int;
      statPrevDeleteNum { ExternalAccessible := 'False'; ExternalVisible := 'False'; ExternalWritable := 'False'} : Int;
      statPrevOut { ExternalAccessible := 'False'; ExternalVisible := 'False'; ExternalWritable := 'False'} : String[60];
      statChangeNotAllowedTimer {InstructionName := 'TON_TIME'; LibVersion := '1.0'; ExternalAccessible := 'False'; ExternalVisible := 'False'; ExternalWritable := 'False'} : TON_TIME;
      statTimerEN { ExternalAccessible := 'False'; ExternalVisible := 'False'; ExternalWritable := 'False'} : Bool;
   END_VAR

   VAR CONSTANT 
      DELAY_TIME : Time := T#3s;
   END_VAR


BEGIN
	//============================================================================================================
	// SIEMENS AG
	// (c)Copyright 2019 All Rights Reserved
	//------------------------------------------------------------------------------------------------------------
	// Library: LCPG
	// Tested with: S7-1500 with FW version V2.1
	// Engineering: TIA Portal V14
	// Restrictions: ---
	// Requirements: S7-1500
	// Functionality: instantiate this once in the program for each recipe setpoint of STRING
	// Support: tech.team.motioncontrol@siemens.com
	//------------------------------------------------------------------------------------------------------------
	// Change log table:
	// Version       Date               Expert in charge    Changes applied
	//  01.01.00     02.01.2019         KB                  Initial Release
	//============================================================================================================
	// Function : CPG_RecipeSetpoint_STRING
	//============================================================================================================
	
	// Language Selection
	#recipeSetpoint.CurrentSetpointName := #recipeSetpoint.SetpointName[#recipeControl.LanguageSelection];
	
	//Recipe Disable Control
	#recipeSetpoint.DisableRecipeControl := #disableRecipeControl;
	
	//Pass through enable bit
	#recipeSetpoint.SetpointChangeEnabled := #enable;
	
	//Set out value to match initial one on first scan
	IF #statFirstScan THEN
	    #recipeSetpoint.CurrentRecipeValue := #recipeSetpoint.RecipeValues[#recipeControl.CurrentRecipeID];
	    #recipeSetpoint.OUT := #recipeSetpoint.RecipeValues[#recipeControl.CurrentRecipeID];
	    #statFirstScan := false;
	END_IF;
	
	
	REGION RECIPE CONTROL
	    // Recipe Control - Change, Save, Copy, Delete, Revert setpoint, Save setpoint
	    IF NOT (#recipeSetpoint.DisableRecipeControl) THEN
	        //Recipe Change command
	        IF #recipeControl.RecipeChangeNum <> #statPrevChangeNum THEN
	            #recipeSetpoint.OUT := #recipeSetpoint.RecipeValues[#recipeControl.CurrentRecipeID];
	            #statPrevChangeNum := #recipeControl.RecipeChangeNum;
	            // Prevents multiple commands from being executed if this instruction is not being scanned
	            #statPrevSaveNum := #recipeControl.RecipeSaveNum;
	            #statPrevCopyNum := #recipeControl.RecipeCopyNum;
	            #statPrevDeleteNum := #recipeControl.RecipeDeleteNum;
	        END_IF;
	        //Recipe Save command
	        IF #recipeControl.RecipeSaveNum <> #statPrevSaveNum THEN
	            #recipeSetpoint.RecipeValues[#recipeControl.RecipeDestinationID] := #recipeSetpoint.OUT;
	            #statPrevSaveNum := #recipeControl.RecipeSaveNum;
	            // Prevents multiple commands from being executed if this instruction is not being scanned
	            #statPrevCopyNum := #recipeControl.RecipeCopyNum;
	            #statPrevDeleteNum := #recipeControl.RecipeDeleteNum;
	        END_IF;
	        //Recipe Copy command
	        IF #recipeControl.RecipeCopyNum <> #statPrevCopyNum THEN
	            #recipeSetpoint.RecipeValues[#recipeControl.RecipeDestinationID] := #recipeSetpoint.RecipeValues[#recipeControl.RecipeSourceID];
	            #statPrevCopyNum := #recipeControl.RecipeCopyNum;
	            // Prevents multiple commands from being executed if this instruction is not being scanned
	            #statPrevDeleteNum := #recipeControl.RecipeDeleteNum;
	        END_IF;
	        //Recipe Delete command
	        IF #recipeControl.RecipeDeleteNum <> #statPrevDeleteNum THEN
	            //edit this line to change the value a deleted recipe defaults to
	            #recipeSetpoint.RecipeValues[#recipeControl.RecipeDestinationID] := ''; 
	            #statPrevDeleteNum := #recipeControl.RecipeDeleteNum;
	        END_IF;
	        //Revert setpoint to saved value
	        IF #recipeSetpoint.RevertSetpoint THEN
	            #recipeSetpoint.OUT := #recipeSetpoint.RecipeValues[#recipeControl.CurrentRecipeID];
	        END_IF;
	        //Detect recipe/setpoint difference
	        IF (#recipeSetpoint.RecipeValues[#recipeControl.CurrentRecipeID] <> #recipeSetpoint.OUT) AND NOT (#recipeControl.RecipeChange) THEN
	            #recipeControl.RecipeSetpointDiff := true;  //signal to recipe control that a setpoint differs
	            #recipeSetpoint.RecipeSetpointDiff := true;
	        ELSE
	            #recipeSetpoint.RecipeSetpointDiff := false;
	        END_IF;
	        //Save setpoint
	        IF #recipeSetpoint.SaveSetpoint THEN
	            #recipeSetpoint.RecipeValues[#recipeControl.CurrentRecipeID] := #recipeSetpoint.OUT;
	        END_IF;
	        
	        //update values stored for current recipe & recipes A, B, & C
	        #recipeSetpoint.CurrentRecipeValue := #recipeSetpoint.RecipeValues[#recipeControl.CurrentRecipeID];
	        #recipeSetpoint.RecipeValueA := #recipeSetpoint.RecipeValues[#recipeControl.RecipeID_A];
	        #recipeSetpoint.RecipeValueB := #recipeSetpoint.RecipeValues[#recipeControl.RecipeID_B];
	        #recipeSetpoint.RecipeValueC := #recipeSetpoint.RecipeValues[#recipeControl.RecipeID_C];
	        
	    ELSE    //if recipe control is disabled, just update counters
	        #recipeSetpoint.RecipeSetpointDiff := false;
	        #statPrevChangeNum := #recipeControl.RecipeChangeNum;
	        #statPrevSaveNum := #recipeControl.RecipeSaveNum;
	        #statPrevCopyNum := #recipeControl.RecipeCopyNum;
	        #statPrevDeleteNum := #recipeControl.RecipeDeleteNum;
	    END_IF;
	END_REGION
	
	
	REGION UPDATE IN VALUE
	    //If ENABLE, then changes to the setpoint value are possible
	    //otherwise, updating the setpoint is not possible via changing RecipeSetpoint.IN
	    IF #enable THEN
	        //Clear status bit
	        #recipeSetpoint.SetpointChangeDisabled := false;
	        
	        // Check for input changed (due to user updating RecipeSetpoint.IN)
	        IF (#recipeSetpoint.IN <> #recipeSetpoint.OUT) AND (#recipeSetpoint.OUT = #statPrevOut) THEN
	            #recipeSetpoint.OUT := #recipeSetpoint.IN;
	        // Check for output changed (due to a recipe change)
	        ELSIF (#recipeSetpoint.IN <> #recipeSetpoint.OUT) AND (#recipeSetpoint.OUT <> #statPrevOut) THEN
	            #recipeSetpoint.IN := #recipeSetpoint.OUT;
	        END_IF;
	        
	    ELSE
	        
	        // If IN changes, revert and display message
	        IF (#recipeSetpoint.IN <> #recipeSetpoint.OUT) OR #recipeSetpoint.RevertSetpoint THEN
	            #recipeSetpoint.IN := #recipeSetpoint.OUT;
	            #statTimerEN := false;
	            #recipeSetpoint.SetpointChangeDisabled := true;
	        END_IF;
	        
	        //display "setpoint changes not allowed" 3 seconds after inputting an invalid change
	        #statChangeNotAllowedTimer(IN := #statTimerEN,
	                               PT := #DELAY_TIME);
	        
	        // Continue to display the status bits for the duration of the timer.
	        IF #recipeSetpoint.SetpointChangeDisabled THEN
	            #statTimerEN := true;
	            #recipeSetpoint.SetpointChangeDisabled :=
	                #recipeSetpoint.SetpointChangeDisabled AND #statTimerEN AND NOT #statChangeNotAllowedTimer.Q;
	        END_IF;
	        
	    END_IF;
	END_REGION
	
	
	REGION Set Outputs
	    IF (#recipeSetpoint.OUT <> #statPrevOut) THEN
	        #statPrevOut := #recipeSetpoint.OUT;
	    END_IF;
	    #out := #recipeSetpoint.OUT;
	    #changeNotAllowed := #recipeSetpoint.SetpointChangeDisabled;
	    #recipeSetpointDifference := #recipeSetpoint.RecipeSetpointDiff;
	    #recipeControlDisabled := #recipeSetpoint.DisableRecipeControl;
	    #changeEnabled := #recipeSetpoint.SetpointChangeEnabled;
	END_REGION
	
	//  -------------- END OF LOGIC -------------------------
	ENO := TRUE;   // Set the ENO output
END_FUNCTION_BLOCK

FUNCTION_BLOCK "BeltConveyor"
{ S7_Optimized_Access := 'TRUE' }
VERSION : 0.1
   VAR_INPUT 
      bx_BoxSensor : Bool;
      bx_BoxReq : Bool;
      ix_CurrentState : DInt;
   END_VAR

   VAR_OUTPUT 
      by_BeltFrd : Bool;
      by_BoxReady : Bool;
      ModuleSts : "CPG_typePackML_ModuleSts";
      iy_SeqStep : Int;
   END_VAR

   VAR 
      i_SeqStep : Int;
   END_VAR


BEGIN
	CASE #ix_CurrentState OF
	    1://Clearing
	        #ModuleSts.sts_Clearing_SC := True;
	    2://Stopped
	        #ModuleSts.sts_Stopping_SC := False;
	        #ModuleSts.sts_Clearing_SC := False;
	    3://Starting
	        #ModuleSts.sts_Starting_SC := True;
	        #iy_SeqStep := #i_SeqStep;
	    4://Idle
	        #ModuleSts.sts_Resetting_SC := False;
	        #i_SeqStep := 0;
	    5://Suspended
	        ;
	    6://Execute
	        #ModuleSts.sts_Starting_SC := False;
	        CASE #i_SeqStep OF
	            0://Start the conveyor, wait the box arrive
	                #by_BeltFrd := True;
	                IF #bx_BoxSensor THEN
	                    #by_BeltFrd := False;
	                    #by_BoxReady := True;
	                    #i_SeqStep := 1;
	                END_IF;
	            1://Wait for the request
	                IF #bx_BoxReq THEN
	                    #by_BeltFrd := True;
	                    #i_SeqStep := 2;
	                END_IF;
	            2://Wait the box leave 
	                IF NOT #bx_BoxSensor THEN
	                    #by_BoxReady := False;
	                    #i_SeqStep := 0;
	                END_IF;
	                ;
	        END_CASE;
	        //#ModuleSts.sts_Execute_SC := True;
	    7://Stopping
	        #ModuleSts.sts_Stopping_SC := True;
	    8://Aborting
	        #ModuleSts.sts_Aborting_SC := True;
	    9://Aborted
	        #ModuleSts.sts_Aborting_SC := False;
	    10://Holding
	        #ModuleSts.sts_Holding_SC := True;
	    11://Held
	        ;
	    12://Unholding
	        ;
	    13://Suspending
	        ;
	    14://Unsuspending
	        ;
	    15://Resetting
	        #ModuleSts.cmd_Reset := False;
	        #ModuleSts.sts_Resetting_SC := True;
	    16://Completing
	        #ModuleSts.sts_Execute_SC := False;
	        #ModuleSts.sts_Completing_SC := True;
	    17://Complete
	        #ModuleSts.sts_Completing_SC := False;
	END_CASE;
	#iy_SeqStep := #i_SeqStep;
END_FUNCTION_BLOCK

FUNCTION_BLOCK "Conveyor"
{ S7_Optimized_Access := 'TRUE' }
VERSION : 0.1
   VAR_INPUT 
      bx_PalletSensor : Bool;
      bx_NextReq : Bool;
      ix_CurrentState : DInt;
   END_VAR

   VAR_OUTPUT 
      by_ConvFrd : Bool;
      by_NextAck : Bool;
      ModuleSts : "CPG_typePackML_ModuleSts";
      iy_SeqStep : Int;
   END_VAR

   VAR 
      i_SeqStep : Int;
   END_VAR


BEGIN
	CASE #ix_CurrentState OF
	    1://Clearing
	        #ModuleSts.sts_Clearing_SC := True;
	    2://Stopped
	        #ModuleSts.sts_Stopping_SC := False;
	        #ModuleSts.sts_Clearing_SC := False;
	    3://Starting
	        #ModuleSts.sts_Starting_SC := True;
	        #iy_SeqStep := #i_SeqStep;
	    4://Idle
	        #ModuleSts.sts_Resetting_SC := False;
	        #i_SeqStep := 0;
	    5://Suspended
	        ;
	    6://Execute
	        #ModuleSts.sts_Starting_SC := False;
	        CASE #i_SeqStep OF
	            0://Check if pallet is present
	                IF #bx_PalletSensor THEN
	                    #i_SeqStep := 2; 
	                ELSIF NOT #bx_PalletSensor THEN
	                    #i_SeqStep := 1;
	                END_IF;
	            1://Run the conveyor
	                #by_ConvFrd := True;
	                IF #bx_PalletSensor THEN
	                    #by_ConvFrd := False;
	                    #i_SeqStep := 2;
	                END_IF;
	            2://Wait req from next module
	                IF #bx_NextReq THEN
	                    #by_NextAck := True;
	                    #by_ConvFrd := True;
	                    #i_SeqStep := 3;
	                END_IF;
	            3://Wait pallet leave
	                IF NOT #bx_PalletSensor THEN
	                    #by_NextAck := False;
	                    #by_ConvFrd := False;
	                    #i_SeqStep := 0;
	                END_IF;
	        END_CASE;
	        //#ModuleSts.sts_Execute_SC := True;
	    7://Stopping
	        #ModuleSts.sts_Stopping_SC := True;
	    8://Aborting
	        #ModuleSts.sts_Aborting_SC := True;
	    9://Aborted
	        #ModuleSts.sts_Aborting_SC := False;
	    10://Holding
	        #ModuleSts.sts_Holding_SC := True;
	    11://Held
	        ;
	    12://Unholding
	        ;
	    13://Suspending
	        ;
	    14://Unsuspending
	        ;
	    15://Resetting
	        #ModuleSts.cmd_Reset := False;
	        #ModuleSts.sts_Resetting_SC := True;
	    16://Completing
	        #ModuleSts.sts_Execute_SC := False;
	        #ModuleSts.sts_Completing_SC := True;
	    17://Complete
	        #ModuleSts.sts_Completing_SC := False;
	END_CASE;
	#iy_SeqStep := #i_SeqStep;
END_FUNCTION_BLOCK

FUNCTION_BLOCK "ConveyorCrossing"
{ S7_Optimized_Access := 'TRUE' }
VERSION : 0.1
   VAR_INPUT 
      bx_PalletSensor : Bool;
      bx_P1_PalletReq : Bool;
      bx_P2_PalletReq : Bool;
      ix_CurrentState : DInt;
   END_VAR

   VAR_OUTPUT 
      by_RollsFrd : Bool;
      by_RollsRev : Bool;
      by_ChainFrd : Bool;
      by_ChainRev : Bool;
      by_P1_Ack : Bool;
      by_P2_Ack : Bool;
      ModuleSts : "CPG_typePackML_ModuleSts";
      iy_SeqStep : Int;
   END_VAR

   VAR 
      i_SeqStep : Int;
   END_VAR


BEGIN
	CASE #ix_CurrentState OF
	    1://Clearing
	        #ModuleSts.sts_Clearing_SC := True;
	    2://Stopped
	        #ModuleSts.sts_Stopping_SC := False;
	        #ModuleSts.sts_Clearing_SC := False;
	    3://Starting
	        #ModuleSts.sts_Starting_SC := True;
	        #iy_SeqStep := #i_SeqStep;
	    4://Idle
	        #ModuleSts.sts_Resetting_SC := False;
	        #i_SeqStep := 0;
	    5://Suspended
	        ;
	    6://Execute
	        #ModuleSts.sts_Starting_SC := False;
	        CASE #i_SeqStep OF
	            0://Wait req
	                IF #bx_P1_PalletReq THEN
	                    #i_SeqStep := 1;
	                ELSIF #bx_P2_PalletReq THEN
	                    #i_SeqStep := 2;
	                END_IF;
	            1://Start the rolls, wait pallet arrive
	                #by_RollsFrd := True;
	                
	               
	        END_CASE;
	        //#ModuleSts.sts_Execute_SC := True;
	    7://Stopping
	        #ModuleSts.sts_Stopping_SC := True;
	    8://Aborting
	        #ModuleSts.sts_Aborting_SC := True;
	    9://Aborted
	        #ModuleSts.sts_Aborting_SC := False;
	    10://Holding
	        #ModuleSts.sts_Holding_SC := True;
	    11://Held
	        ;
	    12://Unholding
	        ;
	    13://Suspending
	        ;
	    14://Unsuspending
	        ;
	    15://Resetting
	        #ModuleSts.cmd_Reset := False;
	        #ModuleSts.sts_Resetting_SC := True;
	    16://Completing
	        #ModuleSts.sts_Execute_SC := False;
	        #ModuleSts.sts_Completing_SC := True;
	    17://Complete
	        #ModuleSts.sts_Completing_SC := False;
	END_CASE;
	#iy_SeqStep := #i_SeqStep;
END_FUNCTION_BLOCK

FUNCTION_BLOCK "PackML_Template"
{ S7_Optimized_Access := 'TRUE' }
VERSION : 0.1
   VAR_INPUT 
      ix_CurrentState : DInt;
   END_VAR

   VAR_OUTPUT 
      ModuleSts : "CPG_typePackML_ModuleSts";
      iy_SeqStep : Int;
   END_VAR

   VAR 
      i_SeqStep : Int;
   END_VAR


BEGIN
	CASE #ix_CurrentState OF
	    1://Clearing
	        #ModuleSts.sts_Clearing_SC := True;
	    2://Stopped
	        #ModuleSts.sts_Stopping_SC := False;
	        #ModuleSts.sts_Clearing_SC := False;
	    3://Starting
	        #ModuleSts.sts_Starting_SC := True;
	        #iy_SeqStep := #i_SeqStep;
	    4://Idle
	        #ModuleSts.sts_Resetting_SC := False;
	        #i_SeqStep := 0;
	    5://Suspended
	        ;
	    6://Execute
	        #ModuleSts.sts_Starting_SC := False;
	        //#ModuleSts.sts_Execute_SC := True;
	    7://Stopping
	        #ModuleSts.sts_Stopping_SC := True;
	    8://Aborting
	        #ModuleSts.sts_Aborting_SC := True;
	    9://Aborted
	        #ModuleSts.sts_Aborting_SC := False;
	    10://Holding
	        #ModuleSts.sts_Holding_SC := True;
	    11://Held
	        ;
	    12://Unholding
	        ;
	    13://Suspending
	        ;
	    14://Unsuspending
	        ;
	    15://Resetting
	        #ModuleSts.cmd_Reset := False;
	        #ModuleSts.sts_Resetting_SC := True;
	    16://Completing
	        #ModuleSts.sts_Execute_SC := False;
	        #ModuleSts.sts_Completing_SC := True;
	    17://Complete
	        #ModuleSts.sts_Completing_SC := False;
	END_CASE;
	#iy_SeqStep := #i_SeqStep;
END_FUNCTION_BLOCK

FUNCTION_BLOCK "Palletizer"
{ S7_Optimized_Access := 'TRUE' }
VERSION : 0.1
   VAR_INPUT 
      bx_PalletSensor1 : Bool;
      bx_PalletSensor2 : Bool;
      bx_ProductsReadyToPush : Bool;
      bx_PusherInPos : Bool;
      bx_TrapdoorInPos : Bool;
      bx_PositionerExtended : Bool;
      bx_LiftMoving : Bool;
      bx_BoxReady : Bool;
      bx_PalletReady : Bool;
      ix_CurrentState : DInt;
   END_VAR

   VAR_OUTPUT 
      by_BeltFrd : Bool;
      by_BeltRev : Bool;
      by_Pusher : Bool;
      by_Positioner : Bool;
      by_Trapdoor : Bool;
      by_LiftUp : Bool;
      by_LiftDown : Bool;
      by_ChainFrd : Bool;
      by_ChainRev : Bool;
      by_BoxReq : Bool;
      by_PalletReq : Bool;
      ModuleSts : "CPG_typePackML_ModuleSts";
      iy_SeqStep : Int;
   END_VAR

   VAR 
      i_SeqStep : Int;
   END_VAR


BEGIN
	CASE #ix_CurrentState OF
	    1://Clearing
	        #ModuleSts.sts_Clearing_SC := True;
	    2://Stopped
	        #ModuleSts.sts_Stopping_SC := False;
	        #ModuleSts.sts_Clearing_SC := False;
	    3://Starting
	        #ModuleSts.sts_Starting_SC := True;
	        #iy_SeqStep := #i_SeqStep;
	    4://Idle
	        #ModuleSts.sts_Resetting_SC := False;
	        #i_SeqStep := 0;
	    5://Suspended
	        ;
	    6://Execute
	        #ModuleSts.sts_Starting_SC := False;
	        CASE #i_SeqStep OF
	            0:
	                ;
	        END_CASE;
	        //#ModuleSts.sts_Execute_SC := True;
	    7://Stopping
	        #ModuleSts.sts_Stopping_SC := True;
	    8://Aborting
	        #ModuleSts.sts_Aborting_SC := True;
	    9://Aborted
	        #ModuleSts.sts_Aborting_SC := False;
	    10://Holding
	        #ModuleSts.sts_Holding_SC := True;
	    11://Held
	        ;
	    12://Unholding
	        ;
	    13://Suspending
	        ;
	    14://Unsuspending
	        ;
	    15://Resetting
	        #ModuleSts.cmd_Reset := False;
	        #ModuleSts.sts_Resetting_SC := True;
	    16://Completing
	        #ModuleSts.sts_Execute_SC := False;
	        #ModuleSts.sts_Completing_SC := True;
	    17://Complete
	        #ModuleSts.sts_Completing_SC := False;
	END_CASE;
	#iy_SeqStep := #i_SeqStep;
END_FUNCTION_BLOCK

